    stRecipe.stUCF.iCapSorterTransporterVolumeOfCapsShow.diDefault:=330;
	stRecipe.stUCF.iCapSorterTransporterVolumeOfCapsShow.diMinLimit:=0;
	stRecipe.stUCF.iCapSorterTransporterVolumeOfCapsShow.diMaxLimit:=10000;

    stRecipe.stUCF.iCapSorterWheelWaitingAfterRotationEmptyTableShow.diDefault:=30;
	stRecipe.stUCF.iCapSorterWheelWaitingAfterRotationEmptyTableShow.diMinLimit:=0;
	stRecipe.stUCF.iCapSorterWheelWaitingAfterRotationEmptyTableShow.diMaxLimit:=1000;

    stRecipe.stUCF.iCapSorterWheelWaitingAfterRotationFullTableShow.diDefault:=20;
	stRecipe.stUCF.iCapSorterWheelWaitingAfterRotationFullTableShow.diMinLimit:=0;
	stRecipe.stUCF.iCapSorterWheelWaitingAfterRotationFullTableShow.diMaxLimit:=1000;
	
    stRecipe.stUCF.iCapSorterWheelWaitingAfterRotationHalfFullTableShow.diDefault:=25;
	stRecipe.stUCF.iCapSorterWheelWaitingAfterRotationHalfFullTableShow.diMinLimit:=0;
	stRecipe.stUCF.iCapSorterWheelWaitingAfterRotationHalfFullTableShow.diMaxLimit:=1000;

    stRecipe.stUCF.lrCapSorterBrush1OnWheelPositionHeightSVShow.lrDefault:=20;
	stRecipe.stUCF.lrCapSorterBrush1OnWheelPositionHeightSVShow.lrMinLimit:=0;
	stRecipe.stUCF.lrCapSorterBrush1OnWheelPositionHeightSVShow.lrMaxLimit:=10000;
	
    stRecipe.stUCF.lrCapSorterBrush2OnWheelPositionHeightSVShow.lrDefault:=16;
	stRecipe.stUCF.lrCapSorterBrush2OnWheelPositionHeightSVShow.lrMinLimit:=0;
	stRecipe.stUCF.lrCapSorterBrush2OnWheelPositionHeightSVShow.lrMaxLimit:=10000;

    stRecipe.stUCF.lrCapSorterFeederMover1InputPositionShow.lrDefault:=0;
	stRecipe.stUCF.lrCapSorterFeederMover1InputPositionShow.lrMinLimit:=-10;
	stRecipe.stUCF.lrCapSorterFeederMover1InputPositionShow.lrMaxLimit:=100;
	
	stRecipe.stUCF.lrCapSorterFeederMover1OutputPositionShow.lrDefault:=1147;
	stRecipe.stUCF.lrCapSorterFeederMover1OutputPositionShow.lrMinLimit:=0;
	stRecipe.stUCF.lrCapSorterFeederMover1OutputPositionShow.lrMaxLimit:=1200;
	
    stRecipe.stUCF.lrCapSorterFeederMover2InputPositionShow.lrDefault:=0;
	stRecipe.stUCF.lrCapSorterFeederMover2InputPositionShow.lrMinLimit:=-10;
	stRecipe.stUCF.lrCapSorterFeederMover2InputPositionShow.lrMaxLimit:=100;
	
    stRecipe.stUCF.lrCapSorterFeederMover2OutputPositionShow.lrDefault:=1147;
	stRecipe.stUCF.lrCapSorterFeederMover2OutputPositionShow.lrMinLimit:=0;
    stRecipe.stUCF.lrCapSorterFeederMover2OutputPositionShow.lrMaxLimit:=1200;
	
    stRecipe.stUCF.lrCapSorterFeederMoverAccelerationShow.lrDefault:=60;
	stRecipe.stUCF.lrCapSorterFeederMoverAccelerationShow.lrMinLimit:=0;
	stRecipe.stUCF.lrCapSorterFeederMoverAccelerationShow.lrMaxLimit:=100;
	
    stRecipe.stUCF.lrCapSorterFeederMoverSpeedShow.lrDefault:=50;
	stRecipe.stUCF.lrCapSorterFeederMoverSpeedShow.lrMinLimit:=1;
	stRecipe.stUCF.lrCapSorterFeederMoverSpeedShow.lrMaxLimit:=100;	
	
    stRecipe.stUCF.lrCapSorterFeederSlotDistanceShow.lrDefault:=150;
	stRecipe.stUCF.lrCapSorterFeederSlotDistanceShow.lrMinLimit:=0;
	stRecipe.stUCF.lrCapSorterFeederSlotDistanceShow.lrMaxLimit:=1000;	
	
    stRecipe.stUCF.lrCapSorterIntermediateBrushPositionHeightSVShow.lrDefault:=33;
	stRecipe.stUCF.lrCapSorterIntermediateBrushPositionHeightSVShow.lrMinLimit:=0;
	stRecipe.stUCF.lrCapSorterIntermediateBrushPositionHeightSVShow.lrMaxLimit:=10000;
	
    stRecipe.stUCF.lrCapSorterIntermediateTransporterWheelAngleShow.lrDefault:=3;
	stRecipe.stUCF.lrCapSorterIntermediateTransporterWheelAngleShow.lrMinLimit:=0;
	stRecipe.stUCF.lrCapSorterIntermediateTransporterWheelAngleShow.lrMaxLimit:=360;

    stRecipe.stUCF.lrCapSorterPreScrewerCartesianCatchZPositionShow.lrDefault:=330;
	stRecipe.stUCF.lrCapSorterPreScrewerCartesianCatchZPositionShow.lrMinLimit:=0;
	stRecipe.stUCF.lrCapSorterPreScrewerCartesianCatchZPositionShow.lrMaxLimit:=1000;

    stRecipe.stUCF.lrCapSorterPreScrewerCatcherCatchingPositionShow.lrDefault:=130;
	stRecipe.stUCF.lrCapSorterPreScrewerCatcherCatchingPositionShow.lrMinLimit:=0;
	stRecipe.stUCF.lrCapSorterPreScrewerCatcherCatchingPositionShow.lrMaxLimit:=1000;	
	
    stRecipe.stUCF.lrCapSorterPreScrewerCatcherHightSVShow.lrDefault:=88;
	stRecipe.stUCF.lrCapSorterPreScrewerCatcherHightSVShow.lrMinLimit:=0;
	stRecipe.stUCF.lrCapSorterPreScrewerCatcherHightSVShow.lrMaxLimit:=1000;
	
    stRecipe.stUCF.lrCapSorterPreScrewerCatcherPlacePositionShow.lrDefault:=70;
	stRecipe.stUCF.lrCapSorterPreScrewerCatcherPlacePositionShow.lrMinLimit:=0;
	stRecipe.stUCF.lrCapSorterPreScrewerCatcherPlacePositionShow.lrMaxLimit:=1000;   
	
    stRecipe.stUCF.lrCapSorterPreScrewerCatcherSpeedShow.lrDefault:=20;
	stRecipe.stUCF.lrCapSorterPreScrewerCatcherSpeedShow.lrMinLimit:=1;
	stRecipe.stUCF.lrCapSorterPreScrewerCatcherSpeedShow.lrMaxLimit:=100;  
	
    stRecipe.stUCF.lrCapSorterPreScrewerPickXMover1PositionShow.lrDefault:=188.8;
	stRecipe.stUCF.lrCapSorterPreScrewerPickXMover1PositionShow.lrMinLimit:=0;
	stRecipe.stUCF.lrCapSorterPreScrewerPickXMover1PositionShow.lrMaxLimit:=1000;	
	
    stRecipe.stUCF.lrCapSorterPreScrewerPickXMover2PositionShow.lrDefault:=260;
	stRecipe.stUCF.lrCapSorterPreScrewerPickXMover2PositionShow.lrMinLimit:=0;
	stRecipe.stUCF.lrCapSorterPreScrewerPickXMover2PositionShow.lrMaxLimit:=1000;	
	
    stRecipe.stUCF.lrCapSorterPreScrewerPickZPositionShow.lrDefault:=418;
	stRecipe.stUCF.lrCapSorterPreScrewerPickZPositionShow.lrMinLimit:=0;
	stRecipe.stUCF.lrCapSorterPreScrewerPickZPositionShow.lrMaxLimit:=1000;	
	
	stRecipe.stUCF.lrCapSorterPreScrewerCapCatcherZPositionShow.lrDefault:=450;
	stRecipe.stUCF.lrCapSorterPreScrewerCapCatcherZPositionShow.lrMinLimit:=0;
	stRecipe.stUCF.lrCapSorterPreScrewerCapCatcherZPositionShow.lrMaxLimit:=1000;
	
    stRecipe.stUCF.lrCapSorterPreScrewerPickerSpeedShow.lrDefault:=10;
	stRecipe.stUCF.lrCapSorterPreScrewerPickerSpeedShow.lrMinLimit:=1;
	stRecipe.stUCF.lrCapSorterPreScrewerPickerSpeedShow.lrMaxLimit:=100;	
	
    stRecipe.stUCF.lrCapSorterPreScrewerPlaceXPositionShow.lrDefault:=485.5;
	stRecipe.stUCF.lrCapSorterPreScrewerPlaceXPositionShow.lrMinLimit:=0;
	stRecipe.stUCF.lrCapSorterPreScrewerPlaceXPositionShow.lrMaxLimit:=1000;	
	
    stRecipe.stUCF.lrCapSorterPreScrewerPlaceZPositionShow.lrDefault:=290;
	stRecipe.stUCF.lrCapSorterPreScrewerPlaceZPositionShow.lrMinLimit:=0;
	stRecipe.stUCF.lrCapSorterPreScrewerPlaceZPositionShow.lrMaxLimit:=1000;	
	
    stRecipe.stUCF.lrCapSorterPreScrewerScrewDistanceShow.lrDefault:=360;
	stRecipe.stUCF.lrCapSorterPreScrewerScrewDistanceShow.lrMinLimit:=0;
	stRecipe.stUCF.lrCapSorterPreScrewerScrewDistanceShow.lrMaxLimit:=1400;	
	
    stRecipe.stUCF.lrCapSorterPreScrewerScrewFindingShow.lrDefault:=0;
	stRecipe.stUCF.lrCapSorterPreScrewerScrewFindingShow.lrMinLimit:=0;
	stRecipe.stUCF.lrCapSorterPreScrewerScrewFindingShow.lrMaxLimit:=1000;	
	
    stRecipe.stUCF.lrCapSorterPreScrewerScrewSpeedShow.lrDefault:=50;
	stRecipe.stUCF.lrCapSorterPreScrewerScrewSpeedShow.lrMinLimit:=1;
	stRecipe.stUCF.lrCapSorterPreScrewerScrewSpeedShow.lrMaxLimit:=100;	
	
    stRecipe.stUCF.lrCapSorterPreScrewerScrewerStartZPositionShow.lrDefault:=305;
	stRecipe.stUCF.lrCapSorterPreScrewerScrewerStartZPositionShow.lrMinLimit:=0;
	stRecipe.stUCF.lrCapSorterPreScrewerScrewerStartZPositionShow.lrMaxLimit:=1000;
	
    stRecipe.stUCF.lrCapSorterPreScrewerStrawCatcherZPositionShow.lrDefault:=286;
	stRecipe.stUCF.lrCapSorterPreScrewerStrawCatcherZPositionShow.lrMinLimit:=0;
	stRecipe.stUCF.lrCapSorterPreScrewerStrawCatcherZPositionShow.lrMaxLimit:=1000;
	
    stRecipe.stUCF.lrCapSorterPreScrewerStrawInsertDistance.lrDefault:=50;
	stRecipe.stUCF.lrCapSorterPreScrewerStrawInsertDistance.lrMinLimit:=0;
	stRecipe.stUCF.lrCapSorterPreScrewerStrawInsertDistance.lrMaxLimit:=1000;	
	
    stRecipe.stUCF.lrCapSorterPreScrewerTopZPositionShow.lrDefault:=470;
	stRecipe.stUCF.lrCapSorterPreScrewerTopZPositionShow.lrMinLimit:=0;
	stRecipe.stUCF.lrCapSorterPreScrewerTopZPositionShow.lrMaxLimit:=1000;
	
    stRecipe.stUCF.lrCapSorterRobotPlace1PositionCShow.lrDefault:=0;
	stRecipe.stUCF.lrCapSorterRobotPlace1PositionCShow.lrMinLimit:=-180;
	stRecipe.stUCF.lrCapSorterRobotPlace1PositionCShow.lrMaxLimit:=180;
	
    stRecipe.stUCF.lrCapSorterRobotPlace1PositionXShow.lrDefault:=0;
	stRecipe.stUCF.lrCapSorterRobotPlace1PositionXShow.lrMinLimit:=-100;
	stRecipe.stUCF.lrCapSorterRobotPlace1PositionXShow.lrMaxLimit:=100;
	
    stRecipe.stUCF.lrCapSorterRobotPlace1PositionYShow.lrDefault:=0;
	stRecipe.stUCF.lrCapSorterRobotPlace1PositionYShow.lrMinLimit:=-100;
	stRecipe.stUCF.lrCapSorterRobotPlace1PositionYShow.lrMaxLimit:=100;
	
    stRecipe.stUCF.lrCapSorterRobotPlace1PositionZShow.lrDefault:=20;
	stRecipe.stUCF.lrCapSorterRobotPlace1PositionZShow.lrMinLimit:=-100;
	stRecipe.stUCF.lrCapSorterRobotPlace1PositionZShow.lrMaxLimit:=100;
	
   	stRecipe.stUCF.lrCapSorterWheelMoveAngleEmptyTableShow.lrDefault:=16;
	stRecipe.stUCF.lrCapSorterWheelMoveAngleEmptyTableShow.lrMinLimit:=0;
	stRecipe.stUCF.lrCapSorterWheelMoveAngleEmptyTableShow.lrMaxLimit:=360;
	
    stRecipe.stUCF.lrCapSorterWheelMoveAngleFullyTableShow.lrDefault:=1;
	stRecipe.stUCF.lrCapSorterWheelMoveAngleFullyTableShow.lrMinLimit:=0;
	stRecipe.stUCF.lrCapSorterWheelMoveAngleFullyTableShow.lrMaxLimit:=360;
	
    stRecipe.stUCF.lrCapSorterWheelMoveAngleHalfFullyTableShow.lrDefault:=6;
	stRecipe.stUCF.lrCapSorterWheelMoveAngleHalfFullyTableShow.lrMinLimit:=0;
	stRecipe.stUCF.lrCapSorterWheelMoveAngleHalfFullyTableShow.lrMaxLimit:=360;
	
    stRecipe.stUCF.udiCapSorterIntermediateTransporterTimeProductOnSensorShow.udiDefault:=800;
	stRecipe.stUCF.udiCapSorterIntermediateTransporterTimeProductOnSensorShow.udiMinLimit:=0;
	stRecipe.stUCF.udiCapSorterIntermediateTransporterTimeProductOnSensorShow.udiMaxLimit:=10000;
	
    stRecipe.stUCF.udiCapSorterTransporterTimeProductOnSensorBeforeBrushShow.udiDefault:=110;
	stRecipe.stUCF.udiCapSorterTransporterTimeProductOnSensorBeforeBrushShow.udiMinLimit:=0;
	stRecipe.stUCF.udiCapSorterTransporterTimeProductOnSensorBeforeBrushShow.udiMaxLimit:=10000;
	
    stRecipe.stUCF.uiCapSorterIndexShow.udiDefault:=8;
	stRecipe.stUCF.uiCapSorterIndexShow.udiMinLimit:=1;
	stRecipe.stUCF.uiCapSorterIndexShow.udiMaxLimit:=100000;
	
	stRecipe.stUCF.lrCapSorterWheelMoveDecelerationEmptyTableShow.lrDefault:=4000;//nie używane
	
	stRecipe.stUCF.lrCapSorterWheelMoveDecelerationFullTableShow.lrDefault:=4000;//nie używane
	
	stRecipe.stUCF.lrCapSorterWheelMoveDecelerationHalfFullTableShow.lrDefault:=4000;//nie używane
	
	stRecipe.stUCF.lrCapSorterWheelMoveSpeedEmptyTableShow.lrDefault:=300;//nie używane
	
	stRecipe.stUCF.lrCapSorterWheelMoveSpeedFullTableShow.lrDefault:=300;//nie używane
	
	stRecipe.stUCF.lrCapSorterWheelMoveSpeedHalfFullTableShow.lrDefault:=300;//nie używane
	
	stRecipe.stUCF.lrCapSorterWheelJerkAngleEmptyTableShow.lrDefault:=10000;//nie używane
	
	stRecipe.stUCF.lrCapSorterWheelJerkAngleFullTableShow.lrDefault:=14000;//nie używane
	
	stRecipe.stUCF.lrCapSorterWheelJerkAngleHalfFullTableShow.lrDefault:=14000;//nie używane
	
	stRecipe.stUCF.lrCapSorterWheelMoveAccelerationEmptyTableShow.lrDefault:=4000;//nie używane
	
	stRecipe.stUCF.lrCapSorterWheelMoveAccelerationFullTableShow.lrDefault:=4000;//nie używane
	
	stRecipe.stUCF.lrCapSorterWheelMoveAccelerationHalfFullTableShow.lrDefault:=4000;//nie używane
	
    stRecipe.stUCF.lrCapSorterPreScrewerScrewJerkShow.lrDefault:=350000;//nie używane
	
	stRecipe.stUCF.lrCapSorterPreScrewerScrewAccelerationShow.lrDefault:=30000;//nie używane
	
	stRecipe.stUCF.lrCapSorterPreScrewerPickerAccelerationShow.lrDefault:=30000;//nie używane
	
	stRecipe.stUCF.lrCapSorterPreScrewerPickerJerkShow.lrDefault:=100000;//nie używane	
	
	stRecipe.stUCF.lrCapSorterPreScrewerGripperOpenPositionShow.lrDefault:=275;//nie używane
	
	stRecipe.stUCF.lrCapSorterPreScrewerCatcherReleseShow.lrDefault:=240;//nie używane
	
	stRecipe.stUCF.lrCapSorterPreScrewerCatcherJerkShow.lrDefault:=100000;//nie używane
	
	stRecipe.stUCF.lrCapSorterPreScrewerCatchAngleOpenSV.lrDefault:=180;//nie używane w ekranie receptur
	
	stRecipe.stUCF.lrCapSorterPreScrewerCatcherAccelerationShow.lrDefault:=40000;// nie używane
	
	stRecipe.stUCF.lrCapSorterPreScrewerBendingDistanceShow.lrDefault:=10;//nie używane
	
	stRecipe.stUCF.lrCapSorterPreScrewerBottleCatch1CloseValueShow.lrDefault:=20600;//nie używane
	
	stRecipe.stUCF.lrCapSorterPreScrewerBottleCatch1OpenValueShow.lrDefault:=43110;//nie używane
	
	stRecipe.stUCF.lrCapSorterPreScrewerBottleCatch2CloseValueShow.lrDefault:=23300;//nie używane
	
	stRecipe.stUCF.lrCapSorterPreScrewerBottleCatch2OpenValueShow.lrDefault:=45548;//nie używane
	
	stRecipe.stUCF.lrCapSorterPreScrewerBottleCatch3CloseValueShow.lrDefault:=21200;//nie uzywane
	
	stRecipe.stUCF.lrCapSorterPreScrewerBottleCatch3OpenValueShow.lrDefault:=44110;//nie używane
	
	stRecipe.stUCF.lrCapSorterPreScrewerBottleCatch4CloseValueShow.lrDefault:=19500;//nie używane
	
	stRecipe.stUCF.lrCapSorterPreScrewerBottleCatch4OpenValueShow.lrDefault:=42487;//nie używane
	
	stRecipe.stUCF.lrCapSorterFeederMoveJerkShow.lrDefault:=370000;//nie używane
	
	stRecipe.stUCF.iCapSorterRobotGripperWatchdogShow.diDefault:=10;//nie używane
	
	stRecipe.stUCF.iCapSorterRobotNumberToolShow.diDefault:=0;//nie używane
	
	stRecipe.stUCF.iCapSorterRobotParalaxCorrectionShow.diDefault:=0;//nie używane
	
	stRecipe.stUCF.iCapSorterIntermediateTransporterManualSpeedShow.diDefault:=30;//nie używane
	
	stRecipe.stUCF.iCapSorterIntermediateBrushManualSpeedShow.diDefault:=30;//nie używane
	
	stRecipe.stUCF.iCapSorterBrush2OnWheelManualSpeedShow.diDefault:=20;//nie używane
	
	stRecipe.stUCF.iCapSorterBrush1OnWheelManualSpeedShow.diDefault:=30;//nie używane
	
	stRecipe.stUCF.lrCapSorterPreScrewerWaitInPlaceTimeShow.lrDefault:=50;//nie używane
	
	stRecipe.stUBF.lrBottleSorterZPickAboveTheBottleSVShow.lrDefault:=0;// nie używane

	stRecipe.stUBF.lrBottleSorterZPickMoveSVShow.lrDefault:=0;// nie używane

	stRecipe.stUBF.uiBottleSorterIndexShow.diDefault:=0;// nie używane
	
	stRecipe.stUBF.lrBottleSorterRemainingTimeToRejectShow.lrDefault:=0;//nie używane
	
	stRecipe.stUBF.lrBottleSorterRemainingTimeToSuctionShow.lrDefault:=0;// nie używane
	
	stRecipe.stUBF.lrBottleSorterSafetyHeightSVShow.lrDefault:=0;// nie używane
	
	stRecipe.stUBF.lrBottleSorterSuckerSuctionTimeShow.lrDefault:=0;// nie używane
	
	stRecipe.stUBF.lrBottleSorterEjectorPulseShow.lrDefault:=0;//nie używane
	
	stRecipe.stUBF.iBottleSorterSupplyTimeThirdConditionSVShow.diDefault:=0;//nie używane
	
	stRecipe.stUBF.iBottleSorterSensorsCountSecondConditionMinSVShow.diDefault:=0;//nie używane
	
	stRecipe.stUBF.iBottleSorterSensorsCountThirdConditionSVShow.diDefault:=0;//nie używane
	
	stRecipe.stUBF.iBottleSorterProductTypeShow.diDefault:=0; //nie używane
	
	stRecipe.stUBL.iLidPuttedCheckProgramShow.diDefault:=0;// nie używane
	
	stRecipe.stUBL.iCapFeederGateBlockingTimeShow.diDefault:=100;// nie używane	
	
    stRecipe.stUBL.iWeight1ActuatorUpDelayShow.diDefault:=0;//nie używane
	
    stRecipe.stUBL.iWeight2ActuatorUpDelayShow.diDefault:=0;//nie używane
	
    stRecipe.stUBL.iWeight3ActuatorUpDelayShow.diDefault:=0;//nie używane
	
    stRecipe.stUBL.iWeight4ActuatorUpDelayShow.diDefault:=0;//nie używane	
	
    stRecipe.stUBL.iWeight5ActuatorUpDelayShow.diDefault:=0;//nie używane	
	
    stRecipe.stUBL.iWeight6ActuatorUpDelayShow.diDefault:=0;//nie używane
	
	stRecipe.stUBL.lrDispencer1SuckValveCloseVolumeShow.lrDefault:=0;//nie używane
	
	stRecipe.stUBL.lrDispencer1DoseValveOpenVolumeShow.lrDefault:=0;//nie używane
	
    stRecipe.stUBL.lrDispencer1LifterAccelerationShow.lrDefault:=15000;//nie używane
	
    stRecipe.stUBL.lrDispencer1LifterDecelerationShow.lrDefault:=15000;//nie używane
	
	stRecipe.stUBL.lrDispencer1LifterVelocityShow.lrDefault:=1050;//nie używane
	
	stRecipe.stUBL.lrDispencer2DoseValveOpenVolumeShow.lrDefault:=0;// nie używane
	
	stRecipe.stUBL.lrDispencer2LifterAccelerationShow.lrDefault:=15000;//nie używane

	stRecipe.stUBL.lrDispencer2LifterDecelerationShow.lrDefault:=15000;//nie używane
		
    stRecipe.stUBL.lrDispencer2LifterVelocityShow.lrDefault:=1050;// nie używane
	
	stRecipe.stUBL.lrDispencer2SuckValveCloseVolumeShow.lrDefault:=0;// nie używane	
	
    stRecipe.stUBL.lrFormWeightShow.lrDefault:=0;//nie używane
	
    stRecipe.stUBL.lrGripperScrewerPressureExhaustLevelShow.lrDefault:=100;//nie używane
		
    stRecipe.stUBL.lrGripperScrewerCatchPressureExhaustLevelShow.lrDefault:=100;//nie używane
	
    stRecipe.stUBL.lrLidPuttedCheckAreaShow.lrDefault:=200;//nie używane
	
    stRecipe.stUBL.lrLidPuttedCheckHeightSVShow.lrDefault:=200;//nie używane
	
    stRecipe.stUBL.lrLidPuttedCheckPositionShow.lrDefault:=200;//nie używane
	
    stRecipe.stUBL.lrMass1DensityShow.lrDefault:=1;//nie używane
	
    stRecipe.stUBL.lrMass2DensityShow.lrDefault:=1;//nie używane
	
    stRecipe.stUBL.lrWeight1MeasurmentCorrectionShow.lrDefault:=0;//nie używane
		
    stRecipe.stUBL.lrWholePackageWeightShow.lrDefault:=0;//nie używane
	
    stRecipe.stUBL.nBottleTransferProgramShow.udiDefault:=0;//nie używane
		
    stRecipe.stUBL.nFormTransportersSlowerVelocitySVShow.udiDefault:=1800;//nie używane
	
    stRecipe.stUBL.nGateAfterWeightTimeFormInsertingShow.lrDefault:=250;//nie używane
	
    stRecipe.stUBL.nGateBeforeDispencersTimeFormInsertingShow.lrDefault:=300;//nie używane
	
    stRecipe.stUBL.nGateRobotTimeFormInsertingShow.lrDefault:=250;//nie używane
END_IF
METH_SortRecipesTable(0);
		udiCurrentIndex																		:=	0;
		wsCurrentCaption1																	:=	"Factory defaults";
		wsCurrentCaption2																	:=	"-";
		METH_SetFactoryDefaults(stPrcRecipe:=stActRecipe);
		udiInitCase										:=	1000;

	1000:
		;

END_CASE
END_ACTION

ACTION ACT_LoadRecipe:
CASE iLoadRecipeCase OF
	0:
				bRecipeLoaded						:=FALSE;
	10:
		IF (iSelectedArrayIndex >=0) THEN 
			IF (aRecipeList[iSelectedArrayIndex].wsRecipeCaption <>"") THEN
				diFileLoadIndex						:=	aRecipeList[iSelectedArrayIndex].udiIndex;
				fbRecipeLoad.sFilePath				:=	CONCAT(CONCAT('C:\Recipes\',DINT_TO_STRING(diFileLoadIndex)),'.CSV');
				fbRecipeLoad.database				:= 	ADR(aRecipeParamsValues);
				fbRecipeLoad.nRows					:= 	udiMaxParamsVariablesCount;
				fbRecipeLoad.nCols					:= 	0;	
				fbRecipeLoad.bExecute				:=	TRUE;
				iLoadRecipeCase						:=	20;
			ELSE
				iLoadRecipeCase				:=	0;
			END_IF
		ELSE
			iLoadRecipeCase					:=	0;
		END_IF
		
	20:
		IF (fbRecipeLoad.bError) THEN
			fbRecipeLoad.bExecute			:=	FALSE;
			iLoadRecipeCase					:=	0;
		END_IF
		IF (fbRecipeLoad.bDone) THEN
			METH_FileStructToRecipeStuct();
			
			wsCurrentCaption1				:=	aRecipeList[diSelectedRecipeFileArrayIndex].wsRecipeCaption;
			wsCurrentCaption2				:=	aRecipeList[diSelectedRecipeFileArrayIndex].wsRecipeDescription;
			udiCurrentIndex					:=	aRecipeList[diSelectedRecipeFileArrayIndex].udiIndex;
			
			fbRecipeLoad.bExecute			:=	FALSE;
			iLoadRecipeCase					:=	0;
			
			bRecipeLoaded					:=	TRUE;
			
			P030_Recipes.bShowRecipeHomingWarning	:=TRUE;
		END_IF
END_CASE
END_ACTION

ACTION ACT_RenameRecipe:
CASE iRenameRecipeCase OF
	0:
		;
	10:
		
		fbRecipeRename.sNetId				:=	'';
		fbRecipeRename.sOldName				:=	CONCAT(CONCAT('C:\Recipes\',UDINT_TO_STRING(udiEditOldIndex)),'.CSV');
		fbRecipeRename.sNewName				:=	CONCAT(CONCAT('C:\Recipes\',UDINT_TO_STRING(udiEditNewIndex)),'.CSV');
		fbRecipeRename.ePath				:= 	PATH_GENERIC;
		fbRecipeRename.tTimeout				:= 	T#3S;
		fbRecipeRename.bExecute				:=	TRUE;
		iRenameRecipeCase					:=	20;
	20:
		IF (fbRecipeRename.bError) THEN
			fbRecipeRename.bExecute			:=	FALSE;
			bEditFail						:=	TRUE;
			wsEditErrorMessage				:=	"Nie udało się zapisać pliku";			
			iRenameRecipeCase				:=	0;
		ELSIF NOT fbRecipeRename.bBusy THEN
			bEditOk							:=	TRUE;
			fbRecipeRename.bExecute			:=	FALSE;
			iRenameRecipeCase				:=	0;			
		END_IF
		
END_CASE
END_ACTION

ACTION ACT_SaveRecipe:
CASE iSaveRecipeCase OF
	0:
		;
	10:
		fbRecipeSave.sFilePath				:=	CONCAT(CONCAT('C:\Recipes\',DINT_TO_STRING(diFileSaveIndex)),'.CSV');
//		fbRecipeSave.database				:= 	ADR(aRecipeParamsValues);
		fbRecipeSave.nRows					:= 	udiMaxParamsVariablesCount;
		fbRecipeSave.nCols					:= 	0;
		fbRecipeSave.bExecute				:=	TRUE;
		iSaveRecipeCase						:=	20;
	20:
		IF (fbRecipeSave.bError OR fbRecipeSave.bDone) THEN
			fbRecipeSave.bExecute			:=	FALSE;
			iSaveRecipeCase					:=	0;
		END_IF
END_CASE
END_ACTION

ACTION ACT_UpdateList:
CASE udiUpdateCase OF
	0:
		;
	10: 
		diRecipeCaptionMaxIndex									:=	-1;
		FOR i:=0 TO udiMaxRecipeCount DO
			IF (aRecipeList[i].bUsed) THEN
				diRecipeCaptionMaxIndex							:=	diRecipeCaptionMaxIndex +1;
//				aRecipeIndexArray[diRecipeCaptionMaxIndex]		:=	UDINT_TO_DINT(i);
				aRecipeCaptionArray[0,diRecipeCaptionMaxIndex]	:=	UDINT_TO_WSTRING(aRecipeList[i].udiIndex);
				aRecipeCaptionArray[1,diRecipeCaptionMaxIndex]	:=	aRecipeList[i].wsRecipeCaption;
				aRecipeCaptionArray[2,diRecipeCaptionMaxIndex]	:=	aRecipeList[i].wsCreateDate;		
			END_IF
		END_FOR
		
		FOR i := DINT_TO_UDINT(diRecipeCaptionMaxIndex +1) TO udiMaxRecipeCount DO
				aRecipeCaptionArray[0,i]						:=	"";
				aRecipeCaptionArray[1,i]						:=	"";
				aRecipeCaptionArray[2,i]						:=	"";	
		END_FOR
		METH_CreateRecipesListStringArray();
		METH_SortRecipesTable(0);
		udiUpdateCase									:=	20;	
	20:
		fbListSave.bExecute								:=	TRUE;
		udiUpdateCase									:=	30;
	30:
		IF (fbListSave.bDone) THEN
			fbListSave.bExecute							:=	FALSE;
			udiUpdateCase								:=	0;
		END_IF
		IF (fbListSave.bError) THEN
			fbListSave.bExecute							:=	FALSE;
			udiUpdateCase								:=	0;
		END_IF

END_CASE

IF bLineSelect THEN
	diSelectedRecipeFileArrayIndex						:= 	METH_FindRecipeArrayIndex(iSelectedArrayIndex);
	wsSelectedCaption									:= 	aRecipeList[diSelectedRecipeFileArrayIndex].wsRecipeCaption;
	udiSelectedRecipeIndex								:=	aRecipeList[diSelectedRecipeFileArrayIndex].udiIndex;	
	bLineSelect											:= 	FALSE;
	
	sProductBitmapId									:= CONCAT('C:\Recipe_photos\RecipeImages.',UDINT_TO_STRING(udiSelectedRecipeIndex));
	sProductBitmapId									:=Concat(sProductBitmapId,'.jpg');
	
END_IF
END_ACTION

METHOD METH_CreateOrClone : BOOL
VAR_INPUT
	bSetDefault				:	BOOL;	
END_VAR
VAR 
	aiCreateDate										:	ARRAY[0..5] OF UINT;
END_VAR

	bAlreadyExist										:=	FALSE;
	bNewRecipeError										:=	FALSE;
	
	IF (wsNewRecipeCaption = "") THEN
		bNewRecipeError									:=	TRUE;
		wsNewRecipeError								:=	"Nazwa nie może być pusta";
	ELSE
		FOR i:= 0 TO udiMaxRecipeCount DO
			IF (aRecipeList[i].bUsed AND (aRecipeList[i].wsRecipeCaption = wsNewRecipeCaption OR aRecipeList[i].udiIndex = udiNewRecipeIndex)) THEN 
				bAlreadyExist							:=	TRUE;
				EXIT;
			END_IF
		END_FOR
		IF (bAlreadyExist) THEN
			bNewRecipeError								:=	TRUE;
			wsNewRecipeError							:=	"Receptura z taką nazwą lub indeksem była dodana wcześnej";
		ELSIF (iSaveRecipeCase >0 OR udiUpdateCase > 0) THEN
			bNewRecipeError								:=	TRUE;
			wsNewRecipeError							:=	"Błąd tworzenia pliku";
		ELSE
			FOR i:= 0 TO udiMaxRecipeCount DO
				IF (NOT aRecipeList[i].bUsed) THEN
					aRecipeList[i].bUsed				:=	TRUE;
					aRecipeList[i].wsRecipeCaption		:=	wsNewRecipeCaption;
					aRecipeList[i].wsRecipeDescription	:=	wsNewRecipeDescription;
					aRecipeList[i].udiIndex				:=	udiNewRecipeIndex;
					
					aiCreateDate[0]		:=	P020_RtcEffectivityOEE.stActualTime.wYear;
					aiCreateDate[1]		:=	P020_RtcEffectivityOEE.stActualTime.wMonth;
					aiCreateDate[2]		:=	P020_RtcEffectivityOEE.stActualTime.wDay;
					aiCreateDate[3]		:=	P020_RtcEffectivityOEE.stActualTime.wHour;
					aiCreateDate[4]		:=	P020_RtcEffectivityOEE.stActualTime.wMinute;
					aiCreateDate[5]		:=	P020_RtcEffectivityOEE.stActualTime.wSecond;
					
					aRecipeList[i].wsCreateDate 		:= METH_DateTimeArray_To_Wstring(aiCreateDate);
					
					IF (bSetDefault) THEN
						METH_SetFactoryDefaults(stPrcRecipe:=stActRecipe);
					END_IF
					METH_RecipeStuctToFileStruct();
					METH_SortRecipesTable(0);				
					diFileSaveIndex						:=	UDINT_TO_INT(udiNewRecipeIndex);
					iSaveRecipeCase						:=	10;
					udiUpdateCase						:=	10;
	
					bNewRecipeOk						:=	TRUE;
					wsNewRecipeError					:=	"";
					EXIT;
				END_IF
			END_FOR
			IF (NOT bNewRecipeOk) THEN
				bNewRecipeError							:=	TRUE;
				wsNewRecipeError						:=	"Nie ma wolnego miejsca w tabeli receptur";
			END_IF
		END_IF
	END_IF
END_METHOD

METHOD METH_CreateRecipesListStringArray : BOOL
VAR

END_VAR

FOR i := 0 TO udiMaxRecipeCount DO
	aRecipeListString[i] := BOOL_TO_STRING(aRecipeList[i].bUsed);
	aRecipeListString[i] := CONCAT(aRecipeListString[i],'|');	
	aRecipeListString[i] := CONCAT(aRecipeListString[i],UDINT_TO_STRING(aRecipeList[i].udiIndex));
	aRecipeListString[i] := CONCAT(aRecipeListString[i],'|');
	aRecipeListString[i] := CONCAT(aRecipeListString[i],WSTRING_TO_STRING(aRecipeList[i].wsRecipeCaption));
	aRecipeListString[i] := CONCAT(aRecipeListString[i],'|');
	aRecipeListString[i] := CONCAT(aRecipeListString[i],WSTRING_TO_STRING(aRecipeList[i].wsRecipeDescription));
	aRecipeListString[i] := CONCAT(aRecipeListString[i],'|');
	aRecipeListString[i] := CONCAT(aRecipeListString[i],WSTRING_TO_STRING(aRecipeList[i].wsCreateDate));
END_FOR
END_METHOD

METHOD METH_DateTimeArray_To_Wstring : WSTRING
VAR_INPUT
	aDate	:	ARRAY[0..5] OF UINT;
END_VAR
VAR 
	wsTmp												:	WSTRING;
END_VAR
IF (aDate[2]<10) THEN
	wsTmp:="0";
END_IF
wsTmp:=WCONCAT(wsTmp,WCONCAT(UINT_TO_WSTRING(aDate[2]),"."));
IF (aDate[1]<10) THEN
	wsTmp:=WCONCAT(wsTmp,"0");
END_IF
wsTmp:=WCONCAT(wsTmp,WCONCAT(UINT_TO_WSTRING(aDate[1]),"."));

IF (aDate[0]<1000) THEN
	wsTmp:=WCONCAT(wsTmp,"0");
ELSIF (aDate[0]<100) THEN
	wsTmp:=WCONCAT(wsTmp,"00");
ELSIF (aDate[0]<10) THEN
	wsTmp:=WCONCAT(wsTmp,"000");
END_IF
wsTmp:=WCONCAT(wsTmp,WCONCAT(UINT_TO_WSTRING(aDate[0])," "));

IF (aDate[3]<10) THEN
	wsTmp:=WCONCAT(wsTmp,"0");
END_IF
wsTmp:=WCONCAT(wsTmp,WCONCAT(UINT_TO_WSTRING(aDate[3]),":"));
IF (aDate[4]<10) THEN
	wsTmp:=WCONCAT(wsTmp,"0");
END_IF
wsTmp:=WCONCAT(wsTmp,WCONCAT(UINT_TO_WSTRING(aDate[4]),"."));
IF (aDate[5]<10) THEN
	wsTmp:=WCONCAT(wsTmp,"0");
END_IF
wsTmp:=WCONCAT(wsTmp,UINT_TO_WSTRING(aDate[5]));
METH_DateTimeArray_To_Wstring:=wsTmp;
END_METHOD

METHOD METH_Edit : BOOL
VAR_INPUT
END_VAR
bEditFail											:=	FALSE;
bEditOk												:=	FALSE;

IF (wsEditNewCaption1 = "") THEN
	bEditFail										:=	TRUE;
	wsEditErrorMessage								:=	"Nazwa nie może być pustą";
ELSE
	FOR i:= 0 TO udiMaxRecipeCount DO
		IF (
			aRecipeList[i].bUsed AND 
			(aRecipeList[i].wsRecipeCaption = wsEditNewCaption1 OR aRecipeList[i].udiIndex =udiEditNewIndex) (*udiEditNewIndex)*) AND
			diSelectedRecipeFileArrayIndex <> UDINT_TO_DINT(i)
			) THEN 
			bEditFail								:=	TRUE;
			wsEditErrorMessage						:=	"Receptura z taką nazwą lub indeksem była dodana wcześniej";	
			RETURN;
		END_IF
	END_FOR
	
	IF (iSelectedArrayIndex >=0) THEN
		IF (diSelectedRecipeFileArrayIndex>=0) THEN
			udiEditOldIndex 													:= 	aRecipeList[diSelectedRecipeFileArrayIndex].udiIndex;
			aRecipeList[diSelectedRecipeFileArrayIndex].udiIndex				:=	udiEditNewIndex;
			aRecipeList[diSelectedRecipeFileArrayIndex].wsRecipeCaption			:=	wsEditNewCaption1;
			aRecipeList[diSelectedRecipeFileArrayIndex].wsRecipeDescription		:=	wsEditNewCaption2;
			IF (udiUpdateCase = 0) THEN
				udiUpdateCase						:=	10;
			END_IF
			IF udiEditOldIndex <> udiEditNewIndex AND iRenameRecipeCase = 0 THEN
				iRenameRecipeCase 					:= 	10;
			END_IF
		END_IF
	END_IF
	IF NOT bEditFail AND iRenameRecipeCase = 0 THEN
		bEditOk											:=	TRUE;		
	END_IF

END_IF
END_METHOD

METHOD METH_FileStructToRecipeStuct : BOOL
VAR_INPUT
END_VAR

VAR
END_VAR
stActRecipe.stUBL.nRecipeIndexShow.diValue															:=						STRING_TO_DINT	(aRecipeParamsValues[0  ]);
stActRecipe.stUBL.iPackageCapTypeShow.diValue														:=						STRING_TO_DINT	(aRecipeParamsValues[1  ]);		
stActRecipe.stUBL.iPackageCapDiameterShow.diValue 													:=						STRING_TO_DINT	(aRecipeParamsValues[2  ]);       
stActRecipe.stUBL.bExEnableShow.bValue 																:=						STRING_TO_BOOL	(aRecipeParamsValues[3  ]);
stActRecipe.stUBL.bBottleFeederEnableShow.bValue													:=						STRING_TO_BOOL	(aRecipeParamsValues[4  ]);
stActRecipe.stUBL.iBottleFeederTurntableVelocitySVShow.udiValue										:=						STRING_TO_UDINT (aRecipeParamsValues[5  ]);
stActRecipe.stUBL.iBottleFeederBottleSensorDelayShow.diValue										:=						STRING_TO_DINT	(aRecipeParamsValues[6  ]);
stActRecipe.stUBL.iBottleFeederFormGateDelayShow.diValue											:=						STRING_TO_DINT	(aRecipeParamsValues[7  ]);
stActRecipe.stUBL.iBottleFeederAllowFormDelayShow.diValue											:=						STRING_TO_DINT	(aRecipeParamsValues[8  ]);
stActRecipe.stUBL.bPucksInserterEnableShow.bValue													:=						STRING_TO_BOOL	(aRecipeParamsValues[9  ]); 
stActRecipe.stUBL.iPucksInserterTurntableVelocitySVShow.udiValue 									:=						STRING_TO_UDINT (aRecipeParamsValues[10 ]);  
stActRecipe.stUBL.iPucksInserterConveyorVelocitySVShow.udiValue										:=						STRING_TO_UDINT (aRecipeParamsValues[11 ]); 
stActRecipe.stUBL.iPucksInserterBottleSensorDelayShow.diValue										:=						STRING_TO_DINT	(aRecipeParamsValues[12 ]);
stActRecipe.stUBL.iPucksInserterFormGateDelayShow.diValue 											:=						STRING_TO_DINT	(aRecipeParamsValues[13 ]);
stActRecipe.stUBL.iPucksInserterAllowFormDelayShow.diValue 											:=						STRING_TO_DINT	(aRecipeParamsValues[14 ]);
stActRecipe.stUBL.lrPucksInserterWheelOffsetShow.lrValue 											:=						STRING_TO_LREAL (aRecipeParamsValues[15 ]);
stActRecipe.stUBL.lrPucksInserterWheelAccelerationShow.lrValue 										:=						STRING_TO_LREAL (aRecipeParamsValues[16 ]);
stActRecipe.stUBL.lrPucksInserterWheelVelocityShow.lrValue 											:=						STRING_TO_LREAL (aRecipeParamsValues[17 ]);
stActRecipe.stUBL.lrPucksInserterHammerHeightSVShow.lrValue 										:=						STRING_TO_LREAL (aRecipeParamsValues[18 ]);
stActRecipe.stUBL.bGateBeforeDispencersEnableShow.bValue											:=						STRING_TO_BOOL	(aRecipeParamsValues[19 ]);
stActRecipe.stUBL.nGateBeforeDispencersTimeFormInsertingShow.lrValue 								:=						STRING_TO_LREAL (aRecipeParamsValues[20 ]);
stActRecipe.stUBL.bGateAfterWeightEnableShow.bValue 												:=						STRING_TO_BOOL	(aRecipeParamsValues[21 ]);
stActRecipe.stUBL.nGateAfterWeightTimeFormInsertingShow.lrValue 									:=						STRING_TO_LREAL (aRecipeParamsValues[22 ]);
stActRecipe.stUBL.bGateRobotEnableShow.bValue       												:=						STRING_TO_BOOL	(aRecipeParamsValues[25 ]);
stActRecipe.stUBL.nGateRobotTimeFormInsertingShow.lrValue											:=						STRING_TO_LREAL (aRecipeParamsValues[26 ]);
stActRecipe.stUBL.bFormsDragingLeftEnableShow.bValue         										:=						STRING_TO_BOOL	(aRecipeParamsValues[27 ]);
stActRecipe.stUBL.lrFormsDragingLeftVelocityShow.lrValue         									:=						STRING_TO_LREAL (aRecipeParamsValues[28 ]);
stActRecipe.stUBL.lrFormsDragingLeftAccelerationShow.lrValue 										:=						STRING_TO_LREAL (aRecipeParamsValues[29 ]);
stActRecipe.stUBL.lrFormsDragingLeftDecelerationShow.lrValue   										:=						STRING_TO_LREAL (aRecipeParamsValues[30 ]);
stActRecipe.stUBL.bFormsDragingRightEnableShow.bValue 												:=						STRING_TO_BOOL	(aRecipeParamsValues[31 ]);
stActRecipe.stUBL.lrFormsDragingRightVelocityShow.lrValue 											:=						STRING_TO_LREAL (aRecipeParamsValues[32 ]);
stActRecipe.stUBL.lrFormsDragingRightAccelerationShow.lrValue 										:=						STRING_TO_LREAL (aRecipeParamsValues[33 ]);
stActRecipe.stUBL.lrFormsDragingRightDecelerationShow.lrValue 										:=						STRING_TO_LREAL (aRecipeParamsValues[34 ]);
stActRecipe.stUBL.bDosingTwoPhasesShow.bValue 	        											:=						STRING_TO_BOOL	(aRecipeParamsValues[35 ]);
stActRecipe.stUBL.lrDispencersLifterReadyPositionShow.lrValue 										:=						STRING_TO_LREAL (aRecipeParamsValues[36 ]);
stActRecipe.stUBL.uiDispencerStartDosingDelayShow.udiValue 											:=						STRING_TO_UDINT (aRecipeParamsValues[37 ]);
stActRecipe.stUBL.bDispencer1EnableShow.bValue 	          											:=						STRING_TO_BOOL	(aRecipeParamsValues[38 ]);
stActRecipe.stUBL.bDispencer2EnableShow.bValue 		  												:=						STRING_TO_BOOL	(aRecipeParamsValues[39 ]);
stActRecipe.stUBL.bDispencer3EnableShow.bValue           											:=						STRING_TO_BOOL	(aRecipeParamsValues[40 ]);
stActRecipe.stUBL.bDispencer4EnableShow.bValue 			       										:=						STRING_TO_BOOL	(aRecipeParamsValues[41 ]);
stActRecipe.stUBL.lrDispencer1DoseVolumeShow.lrValue 				   								:=						STRING_TO_LREAL (aRecipeParamsValues[42 ]);
stActRecipe.stUBL.lrDispencer1Phase1VolumeShow.lrValue	           									:=						STRING_TO_LREAL (aRecipeParamsValues[43 ]);
stActRecipe.stUBL.lrDispencer1Phase2VolumeShow.lrValue 	       										:=						STRING_TO_LREAL (aRecipeParamsValues[44 ]);
stActRecipe.stUBL.lrDispencer1Phase1VelocityShow.lrValue 	       									:=						STRING_TO_LREAL (aRecipeParamsValues[45 ]);
stActRecipe.stUBL.lrDispencer1Phase2VelocityShow.lrValue 											:=						STRING_TO_LREAL (aRecipeParamsValues[46 ]);
stActRecipe.stUBL.lrDispencer1Phase3VelocityShow.lrValue 		   									:=						STRING_TO_LREAL (aRecipeParamsValues[47 ]);
stActRecipe.stUBL.lrDispencer1SuckVelocityShow.lrValue   											:=						STRING_TO_LREAL (aRecipeParamsValues[48 ]);
stActRecipe.stUBL.lrDispencer1Phase1AccelerationShow.lrValue 										:=						STRING_TO_LREAL (aRecipeParamsValues[49 ]);
stActRecipe.stUBL.lrDispencer1Phase2AccelerationShow.lrValue 	  									:=						STRING_TO_LREAL (aRecipeParamsValues[50 ]);
stActRecipe.stUBL.lrDispencer1Phase3AccelerationShow.lrValue 	   									:=						STRING_TO_LREAL (aRecipeParamsValues[51 ]);
stActRecipe.stUBL.lrDispencer1SuckAccelerationShow.lrValue  										:=						STRING_TO_LREAL (aRecipeParamsValues[52 ]);
stActRecipe.stUBL.lrDispencer1Phase1DecelerationShow.lrValue        								:=						STRING_TO_LREAL (aRecipeParamsValues[53 ]);
stActRecipe.stUBL.lrDispencer1Phase2DecelerationShow.lrValue 										:=						STRING_TO_LREAL (aRecipeParamsValues[54 ]);
stActRecipe.stUBL.lrDispencer1Phase3DecelerationShow.lrValue 	   									:=						STRING_TO_LREAL (aRecipeParamsValues[55 ]);
stActRecipe.stUBL.udiDispencer1DosingDoneDelayTimeShow.udiValue 									:=						STRING_TO_UDINT (aRecipeParamsValues[56 ]);
stActRecipe.stUBL.lrDispencer1SuckValveOpenVolumeShow.lrValue 										:=						STRING_TO_LREAL (aRecipeParamsValues[57 ]);
stActRecipe.stUBL.lrDispencer1SuckValveOpenTimeDelayShow.lrValue 									:=						STRING_TO_LREAL (aRecipeParamsValues[58 ]);
stActRecipe.stUBL.lrDispencer1SuckValveCloseVolumeShow.lrValue 										:=						STRING_TO_LREAL (aRecipeParamsValues[59 ]);
stActRecipe.stUBL.lrDispencer1SuckValveCloseTimeDelayShow.lrValue 									:=						STRING_TO_LREAL (aRecipeParamsValues[60 ]);
stActRecipe.stUBL.lrDispencer1DoseValveOpenVolumeShow.lrValue    									:=						STRING_TO_LREAL (aRecipeParamsValues[61 ]);
stActRecipe.stUBL.lrDispencer1DoseValveOpenTimeAccShow.lrValue   									:=						STRING_TO_LREAL (aRecipeParamsValues[62 ]);
stActRecipe.stUBL.lrDispencer1DoseValveCloseVolumeShow.lrValue    									:=						STRING_TO_LREAL (aRecipeParamsValues[63 ]);
stActRecipe.stUBL.lrDispencer1DoseValveCloseTimeDecShow.lrValue 									:=						STRING_TO_LREAL (aRecipeParamsValues[64 ]);
stActRecipe.stUBL.lrDispencer1DoseSuckingVolumeShow.lrValue 										:=						STRING_TO_LREAL (aRecipeParamsValues[65 ]);
stActRecipe.stUBL.lrDispencer1DoseSuckingTimeDelayShow.lrValue 										:=						STRING_TO_LREAL (aRecipeParamsValues[66 ]);
stActRecipe.stUBL.bDispencer1DoseSuckingShow.bValue 			       								:=						STRING_TO_BOOL	(aRecipeParamsValues[67 ]);
stActRecipe.stUBL.bDispencer1LiftSynchroPh1Show.bValue 												:=						STRING_TO_BOOL	(aRecipeParamsValues[68 ]);
stActRecipe.stUBL.bDispencer1LiftSynchroPh2Show.bValue 			   									:=						STRING_TO_BOOL	(aRecipeParamsValues[69 ]);
stActRecipe.stUBL.bDispencer1LiftSynchroPh3Show.bValue 		       									:=						STRING_TO_BOOL	(aRecipeParamsValues[70 ]);
stActRecipe.stUBL.lrDispencer1LifterStartDosePositionShow.lrValue									:=						STRING_TO_LREAL (aRecipeParamsValues[71 ]);
stActRecipe.stUBL.lrDispencer1LifterStopDosePositionShow.lrValue 									:=						STRING_TO_LREAL (aRecipeParamsValues[72 ]);
stActRecipe.stUBL.lrDispencer1LifterVelocityShow.lrValue            								:=						STRING_TO_LREAL (aRecipeParamsValues[73 ]);
stActRecipe.stUBL.lrDispencer1LifterAccelerationShow.lrValue        								:=						STRING_TO_LREAL (aRecipeParamsValues[74 ]);
stActRecipe.stUBL.lrDispencer1LifterDecelerationShow.lrValue 		    							:=						STRING_TO_LREAL (aRecipeParamsValues[75 ]);
stActRecipe.stUBL.lrDispencer2DoseVolumeShow.lrValue	            								:=						STRING_TO_LREAL (aRecipeParamsValues[76 ]);
stActRecipe.stUBL.lrDispencer2Phase1VolumeShow.lrValue 			    								:=						STRING_TO_LREAL (aRecipeParamsValues[77 ]);
stActRecipe.stUBL.lrDispencer2Phase2VolumeShow.lrValue 			    								:=						STRING_TO_LREAL (aRecipeParamsValues[78 ]);
stActRecipe.stUBL.lrDispencer2Phase1VelocityShow.lrValue 		    								:=						STRING_TO_LREAL (aRecipeParamsValues[79 ]);
stActRecipe.stUBL.lrDispencer2Phase2VelocityShow.lrvalue 		    								:=						STRING_TO_LREAL (aRecipeParamsValues[80 ]);
stActRecipe.stUBL.lrDispencer2Phase3VelocityShow.lrValue 		    								:=						STRING_TO_LREAL (aRecipeParamsValues[81 ]);
stActRecipe.stUBL.lrDispencer2SuckVelocityShow.lrValue     											:=						STRING_TO_LREAL (aRecipeParamsValues[82 ]);
stActRecipe.stUBL.lrDispencer2Phase1AccelerationShow.lrValue 	        							:=						STRING_TO_LREAL (aRecipeParamsValues[83 ]);
stActRecipe.stUBL.lrDispencer2Phase2AccelerationShow.lrValue 	        							:=						STRING_TO_LREAL (aRecipeParamsValues[84 ]);
stActRecipe.stUBL.lrDispencer2Phase3AccelerationShow.lrValue 		    							:=						STRING_TO_LREAL (aRecipeParamsValues[85 ]);
stActRecipe.stUBL.lrDispencer2SuckAccelerationShow.lrValue   										:=						STRING_TO_LREAL (aRecipeParamsValues[86 ]);
stActRecipe.stUBL.lrDispencer2Phase1DecelerationShow.lrValue 										:=						STRING_TO_LREAL (aRecipeParamsValues[87 ]);
stActRecipe.stUBL.lrDispencer2Phase2DecelerationShow.lrValue 										:=						STRING_TO_LREAL (aRecipeParamsValues[88 ]);
stActRecipe.stUBL.lrDispencer2Phase3DecelerationShow.lrValue 										:=						STRING_TO_LREAL (aRecipeParamsValues[89 ]);
stActRecipe.stUBL.udiDispencer2DosingDoneDelayTimeShow.udiValue 									:=						STRING_TO_UDINT (aRecipeParamsValues[90 ]);
stActRecipe.stUBL.lrDispencer2SuckValveOpenVolumeShow.lrValue 										:=						STRING_TO_LREAL (aRecipeParamsValues[91 ]);
stActRecipe.stUBL.lrDispencer2SuckValveOpenTimeDelayShow.lrValue 									:=						STRING_TO_LREAL (aRecipeParamsValues[92 ]);
stActRecipe.stUBL.lrDispencer2SuckValveCloseVolumeShow.lrValue										:=						STRING_TO_LREAL (aRecipeParamsValues[93 ]);
stActRecipe.stUBL.lrDispencer2SuckValveCloseTimeDelayShow.lrValue 									:=						STRING_TO_LREAL (aRecipeParamsValues[94 ]);
stActRecipe.stUBL.lrDispencer2DoseValveOpenVolumeShow.lrValue 										:=						STRING_TO_LREAL (aRecipeParamsValues[95 ]);
stActRecipe.stUBL.lrDispencer2DoseValveOpenTimeAccShow.lrValue 										:=						STRING_TO_LREAL (aRecipeParamsValues[96 ]);
stActRecipe.stUBL.lrDispencer2DoseValveCloseVolumeShow.lrValue 										:=						STRING_TO_LREAL (aRecipeParamsValues[97 ]);
stActRecipe.stUBL.lrDispencer2DoseValveCloseTimeDecShow.lrValue										:=						STRING_TO_LREAL (aRecipeParamsValues[98 ]);
stActRecipe.stUBL.lrDispencer2DoseSuckingVolumeShow.lrValue	    									:=						STRING_TO_LREAL (aRecipeParamsValues[99 ]);
stActRecipe.stUBL.lrDispencer2DoseSuckingTimeDelayShow.lrValue										:=						STRING_TO_LREAL (aRecipeParamsValues[100]);
stActRecipe.stUBL.bDispencer2DoseSuckingShow.bValue 	            								:=						STRING_TO_BOOL	(aRecipeParamsValues[101]);
stActRecipe.stUBL.bDispencer2LiftSynchroPh1Show.bValue 	        									:=						STRING_TO_BOOL	(aRecipeParamsValues[102]);
stActRecipe.stUBL.bDispencer2LiftSynchroPh2Show.bValue 	        									:=						STRING_TO_BOOL	(aRecipeParamsValues[103]);
stActRecipe.stUBL.bDispencer2LiftSynchroPh3Show.bValue 	        									:=						STRING_TO_BOOL	(aRecipeParamsValues[104]);
stActRecipe.stUBL.lrDispencer2LifterStartDosePositionShow.lrValue									:=						STRING_TO_LREAL (aRecipeParamsValues[105]);
stActRecipe.stUBL.lrDispencer2LifterStopDosePositionShow.lrValue 									:=						STRING_TO_LREAL (aRecipeParamsValues[106]);
stActRecipe.stUBL.lrDispencer2LifterVelocityShow.lrValue        									:=						STRING_TO_LREAL (aRecipeParamsValues[107]);
stActRecipe.stUBL.lrDispencer2LifterAccelerationShow.lrValue 										:=						STRING_TO_LREAL (aRecipeParamsValues[108]);
stActRecipe.stUBL.lrDispencer2LifterDecelerationShow.lrValue 	    								:=						STRING_TO_LREAL (aRecipeParamsValues[109]);
stActRecipe.stUBL.bDispencersCatchEnableShow.bValue             									:=				   		STRING_TO_BOOL	(aRecipeParamsValues[110]); 	
stActRecipe.stUBL.bDispencersCatchMaxPressureShow.bValue          									:=			   			STRING_TO_BOOL	(aRecipeParamsValues[111]);
stActRecipe.stUBL.lrDispencersCatchHeightSVShow.lrValue												:=						STRING_TO_LREAL (aRecipeParamsValues[112]);	
stActRecipe.stUBL.lrDispencersCatch1ClosedValueShow.lrValue          								:=						STRING_TO_LREAL (aRecipeParamsValues[113]);	
stActRecipe.stUBL.lrDispencersCatch1OpenValueShow.lrValue          									:=						STRING_TO_LREAL (aRecipeParamsValues[114]); 
stActRecipe.stUBL.lrDispencersCatch2ClosedValueShow.lrValue       									:=						STRING_TO_LREAL (aRecipeParamsValues[115]); 
stActRecipe.stUBL.lrDispencersCatch2OpenValueShow.lrValue	    									:=						STRING_TO_LREAL (aRecipeParamsValues[116]);	
stActRecipe.stUBL.lrDispencersCatch3ClosedValueShow.lrValue         								:=						STRING_TO_LREAL (aRecipeParamsValues[117]);
stActRecipe.stUBL.lrDispencersCatch3OpenValueShow.lrValue           								:=						STRING_TO_LREAL (aRecipeParamsValues[118]);	
stActRecipe.stUBL.lrDispencersCatch4ClosedValueShow.lrValue         								:=						STRING_TO_LREAL (aRecipeParamsValues[119]);	
stActRecipe.stUBL.lrDispencersCatch4OpenValueShow.lrValue											:=						STRING_TO_LREAL (aRecipeParamsValues[120]); 
stActRecipe.stUBL.lrDispencersCatchToleranceShow.lrValue 	        								:=						STRING_TO_LREAL (aRecipeParamsValues[121]); 	
stActRecipe.stUBL.bTank1MixerEnableShow.bValue    													:=						STRING_TO_BOOL	(aRecipeParamsValues[122]);
stActRecipe.stUBL.bTankHeatingEnableShow.bValue   													:=						STRING_TO_BOOL	(aRecipeParamsValues[123]);
stActRecipe.stUBL.iTankHeatingTempSVShow.diValue  													:=				        STRING_TO_DINT  (aRecipeParamsValues[124]);
stActRecipe.stUBL.bTank1PressureEnableShow.bValue													:=				        STRING_TO_BOOL  (aRecipeParamsValues[125]);
stActRecipe.stUBL.bTank1SupplyPumpEnableShow.bValue                             					:=                      STRING_TO_BOOL  (aRecipeParamsValues[126]);
stActRecipe.stUBL.bTank2SupplyPumpEnableShow.bValue                             					:=                      STRING_TO_BOOL  (aRecipeParamsValues[127]);
stActRecipe.stUBL.uTank1LevelSetpointShow.udiValue                              					:=                      STRING_TO_UDINT (aRecipeParamsValues[128]);
stActRecipe.stUBL.uTank2LevelSetpointShow.udiValue                              					:=                      STRING_TO_UDINT (aRecipeParamsValues[129]);
stActRecipe.stUBL.bTank1LevelSignalInvertShow.bValue 	                        					:=                      STRING_TO_BOOL  (aRecipeParamsValues[130]);
stActRecipe.stUBL.bTank2LevelSignalInvertShow.bValue 	                        					:=                      STRING_TO_BOOL  (aRecipeParamsValues[131]);
stActRecipe.stUBL.bWeight1EnableShow.bValue                                     					:=       				STRING_TO_BOOL  (aRecipeParamsValues[132]);
stActRecipe.stUBL.lrWeightMassSVShow.lrValue	                                					:=       				STRING_TO_LREAL (aRecipeParamsValues[133]);
stActRecipe.stUBL.iWeight1ActuatorUpDelayShow.diValue 												:=			            STRING_TO_DINT  (aRecipeParamsValues[134]);
stActRecipe.stUBL.iWeight2ActuatorUpDelayShow.diValue                           					:=                      STRING_TO_DINT  (aRecipeParamsValues[135]);
stActRecipe.stUBL.iWeight3ActuatorUpDelayShow.diValue                           					:=                      STRING_TO_DINT  (aRecipeParamsValues[136]);
stActRecipe.stUBL.iWeight4ActuatorUpDelayShow.diValue                           					:=                      STRING_TO_DINT  (aRecipeParamsValues[137]);
stActRecipe.stUBL.iWeight5ActuatorUpDelayShow.diValue                           					:=                      STRING_TO_DINT  (aRecipeParamsValues[138]);
stActRecipe.stUBL.iWeight6ActuatorUpDelayShow.diValue                           					:=                      STRING_TO_DINT  (aRecipeParamsValues[139]);
stActRecipe.stUBL.lrFormWeightShow.lrValue                                      					:=						STRING_TO_LREAL (aRecipeParamsValues[140]);
stActRecipe.stUBL.lrMass1DensityShow.lrValue                                    					:=						STRING_TO_LREAL (aRecipeParamsValues[141]);
stActRecipe.stUBL.lrMass2DensityShow.lrValue                                    					:=						STRING_TO_LREAL (aRecipeParamsValues[142]);
stActRecipe.stUBL.lrCupWeightShow.lrValue                                       					:=						STRING_TO_LREAL (aRecipeParamsValues[143]);
stActRecipe.stUBL.lrWholePackageWeightShow.lrValue 	                            					:=					    STRING_TO_LREAL (aRecipeParamsValues[144]);
stActRecipe.stUBL.lrWeight1MeasurmentCorrectionShow.lrValue	                    					:=					    STRING_TO_LREAL (aRecipeParamsValues[145]);
stActRecipe.stUBL.bDispencer1WeightCorrectionEnableShow.bValue                  					:=					    STRING_TO_BOOL  (aRecipeParamsValues[146]);
stActRecipe.stUBL.bDispencer2WeightCorrectionEnableShow.bValue                  					:=					    STRING_TO_BOOL  (aRecipeParamsValues[147]);
stActRecipe.stUBL.bDispencer3WeightCorrectionEnableShow.bValue                  					:=					    STRING_TO_BOOL  (aRecipeParamsValues[148]);
stActRecipe.stUBL.bDispencer4WeightCorrectionEnableShow.bValue                  					:=					    STRING_TO_BOOL  (aRecipeParamsValues[149]);
stActRecipe.stUBL.lrWeightUpperToleranceShow.lrValue                            					:=					    STRING_TO_LREAL (aRecipeParamsValues[150]);
stActRecipe.stUBL.lrWeightLowerToleranceShow.lrValue                            					:=					    STRING_TO_LREAL (aRecipeParamsValues[151]);
stActRecipe.stUBL.iWeightCorrectionNumberOfSamplesShow.udiValue                 					:=					    STRING_TO_UDINT (aRecipeParamsValues[152]);
stActRecipe.stUBL.bLidFeederEnableShow.bValue                 										:=						STRING_TO_BOOL  (aRecipeParamsValues[153]);
stActRecipe.stUBL.bLidFeederHeaterEnableShow.bValue                             					:=					    STRING_TO_BOOL  (aRecipeParamsValues[154]);
stActRecipe.stUBL.lrLidFeederHeightPosSVShow.lrValue                            					:=					    STRING_TO_LREAL (aRecipeParamsValues[155]);
stActRecipe.stUBL.iLidFeederHeatingTimeShow.diValue                             					:=					    STRING_TO_DINT  (aRecipeParamsValues[156]);
stActRecipe.stUBL.iLidFeederTempHisteresisShow.diValue                          					:=					    STRING_TO_DINT  (aRecipeParamsValues[157]);
stActRecipe.stUBL.iLidFeeder1TempSVShow.diValue 	                            					:=					    STRING_TO_DINT  (aRecipeParamsValues[158]);
stActRecipe.stUBL.iLidFeeder2TempSVShow.diValue 	                            					:=					    STRING_TO_DINT  (aRecipeParamsValues[159]);
stActRecipe.stUBL.bLidFeederDragingStationEnableShow.bValue 	                					:=                      STRING_TO_BOOL  (aRecipeParamsValues[160]);
stActRecipe.stUBL.lrLidFeederDragingStationVelocityShow.lrValue	                					:=                      STRING_TO_LREAL (aRecipeParamsValues[161]);
stActRecipe.stUBL.lrLidFeederDragingStationAccelerationShow.lrValue	            					:=                      STRING_TO_LREAL (aRecipeParamsValues[162]);
stActRecipe.stUBL.lrLidFeederDragingStationDecelerationShow.lrValue	            					:=                      STRING_TO_LREAL (aRecipeParamsValues[163]);
stActRecipe.stUBL.bLidPuttedCheckEnableShow.bValue                              					:=                      STRING_TO_BOOL  (aRecipeParamsValues[164]);
stActRecipe.stUBL.lrLidPuttedCheckHeightSVShow.lrValue                          					:=                      STRING_TO_LREAL (aRecipeParamsValues[165]);
stActRecipe.stUBL.lrLidPuttedCheckPositionShow.lrValue                          					:=                      STRING_TO_LREAL (aRecipeParamsValues[166]);
stActRecipe.stUBL.lrLidPuttedCheckAreaShow.lrValue                              					:=                      STRING_TO_LREAL (aRecipeParamsValues[167]);
stActRecipe.stUBL.iLidPuttedCheckProgramShow.diValue                            					:=      				STRING_TO_DINT  (aRecipeParamsValues[168]);
stActRecipe.stUBL.bLidSealerEnableShow.bValue                                   					:=      				STRING_TO_BOOL  (aRecipeParamsValues[169]);
stActRecipe.stUBL.bLidSealerHeaterEnableShow.bValue 	                        					:=      				STRING_TO_BOOL  (aRecipeParamsValues[170]);
stActRecipe.stUBL.iLidSealerHeatingTimeShow.diValue	                            					:=      				STRING_TO_DINT  (aRecipeParamsValues[171]);
stActRecipe.stUBL.lrLidSealerPressureShow.lrValue                               					:=      				STRING_TO_LREAL (aRecipeParamsValues[172]);
stActRecipe.stUBL.lrLidSealerHeightPosSVShow.lrValue                            					:=      				STRING_TO_LREAL (aRecipeParamsValues[173]);
stActRecipe.stUBL.iLidSealerTempHisteresisShow.diValue                          					:=      				STRING_TO_DINT  (aRecipeParamsValues[174]);
stActRecipe.stUBL.iLidSealer1TempSVShow.diValue 	                            					:=      				STRING_TO_DINT  (aRecipeParamsValues[175]);
stActRecipe.stUBL.iLidSealer2TempSVShow.diValue 	                            					:=      				STRING_TO_DINT  (aRecipeParamsValues[176]);
stActRecipe.stUBL.bLidSealerDragingStationEnableShow.bValue                     					:=      		        STRING_TO_BOOL  (aRecipeParamsValues[177]);
stActRecipe.stUBL.lrLidSealerDragingStationVelocityShow.lrValue 	            					:=      				STRING_TO_LREAL (aRecipeParamsValues[178]);
stActRecipe.stUBL.lrLidSealerDragingStationAccelerationShow.lrValue	            					:=      				STRING_TO_LREAL (aRecipeParamsValues[179]);
stActRecipe.stUBL.lrLidSealerDragingStationDecelerationShow.lrValue	            					:=      				STRING_TO_LREAL (aRecipeParamsValues[180]);
stActRecipe.stUBL.bCapFeederGateEnableShow.bValue 	                            					:=      				STRING_TO_BOOL  (aRecipeParamsValues[181]);
stActRecipe.stUBL.iCapFeederGateBlockingTimeShow.diValue 	                    					:=      				STRING_TO_DINT  (aRecipeParamsValues[182]);
stActRecipe.stUBL.bCapFeederEnableShow.bValue                                   					:=      				STRING_TO_BOOL  (aRecipeParamsValues[183]);
stActRecipe.stUBL.lrCapFeederHeightPosSVShow.lrValue                            					:=                      STRING_TO_LREAL (aRecipeParamsValues[184]);
stActRecipe.stUBL.iCapFeederTimeDelayOnShow.diValue                             					:=                      STRING_TO_DINT  (aRecipeParamsValues[185]);
stActRecipe.stUBL.iCapFeederTimeDelayOffShow.diValue                            					:=                      STRING_TO_DINT  (aRecipeParamsValues[186]);
stActRecipe.stUBL.iCapFeederTimeToEmptySleeveErrorShow.diValue                  					:=                      STRING_TO_DINT  (aRecipeParamsValues[187]);
stActRecipe.stUBL.bCapSorterOnlyWeightOKEnableShow.bValue                       					:=                      STRING_TO_BOOL  (aRecipeParamsValues[188]);
stActRecipe.stUBL.bCapSorterDragEnableShow.bValue                               					:=                      STRING_TO_BOOL  (aRecipeParamsValues[189]);
stActRecipe.stUBL.lrCapSorterDragVelocityShow.lrValue                           					:=                      STRING_TO_LREAL (aRecipeParamsValues[190]);
stActRecipe.stUBL.lrCapSorterDragAccelerationShow.lrValue 	                    					:=                      STRING_TO_LREAL (aRecipeParamsValues[191]);
stActRecipe.stUBL.lrCapSorterDragDecelerationShow.lrValue 	                    					:=                      STRING_TO_LREAL (aRecipeParamsValues[192]);
stActRecipe.stUBL.bCapPuttedCheckEnableShow.bValue                              					:=                      STRING_TO_BOOL  (aRecipeParamsValues[193]);
stActRecipe.stUBL.lrCapPuttedCheckHeightPosSVShow.lrValue 	                    					:=                      STRING_TO_LREAL (aRecipeParamsValues[194]);
stActRecipe.stUBL.bGripperScrewer1EnableShow.bValue 	                        					:=                      STRING_TO_BOOL  (aRecipeParamsValues[195]);
stActRecipe.stUBL.lrGripperScrewingTightTorqueShow.lrValue                      					:=                      STRING_TO_LREAL (aRecipeParamsValues[196]);
stActRecipe.stUBL.bGripperScrewer2EnableShow.bValue 	                        					:=                      STRING_TO_BOOL  (aRecipeParamsValues[197]);
stActRecipe.stUBL.lrGripperScrewing2TightTorqueShow.lrValue	                    					:=                      STRING_TO_LREAL (aRecipeParamsValues[198]);
stActRecipe.stUBL.iGripperScrewer1ToolShow.diValue                              					:=                      STRING_TO_DINT  (aRecipeParamsValues[199]);
stActRecipe.stUBL.lrGripperScrewer1VelocityShow.lrValue                         					:=                      STRING_TO_LREAL (aRecipeParamsValues[200]);
stActRecipe.stUBL.nGripperScrewer1TightTimeShow.diValue	                        					:=                      STRING_TO_DINT  (aRecipeParamsValues[201]);
stActRecipe.stUBL.iGripperScrewer1StartDelayShow.diValue	                    					:=                      STRING_TO_DINT  (aRecipeParamsValues[202]);
stActRecipe.stUBL.lrGripperScrewerReadyPositionShow.lrValue 	                					:=                      STRING_TO_LREAL (aRecipeParamsValues[203]);
stActRecipe.stUBL.lrGripperScrewerPushingCapPositionShow.lrValue 	            					:=                      STRING_TO_LREAL (aRecipeParamsValues[204]);
stActRecipe.stUBL.lrGripperScrewerScrewingCapPositionShow.lrValue               					:=                      STRING_TO_LREAL (aRecipeParamsValues[205]);
stActRecipe.stUBL.lrGripperScrewerPressureShow.lrValue                          					:=                      STRING_TO_LREAL (aRecipeParamsValues[206]);
stActRecipe.stUBL.lrGripperScrewerCatchPressureShow.lrValue 	                					:=                      STRING_TO_LREAL (aRecipeParamsValues[207]);
stActRecipe.stUBL.lrDispencerCatchPressureShow.lrValue                          					:=                      STRING_TO_LREAL (aRecipeParamsValues[208]);
stActRecipe.stUBL.lrGripperScrewerPressureExhaustLevelShow.lrValue              					:=                      STRING_TO_LREAL (aRecipeParamsValues[209]);
stActRecipe.stUBL.lrGripperScrewerCatchPressureExhaustLevelShow.lrValue         					:=                      STRING_TO_LREAL (aRecipeParamsValues[210]);
stActRecipe.stUBL.lrGripperScrewerTurnoversToFullScrewedShow.lrValue 	        					:=                      STRING_TO_LREAL (aRecipeParamsValues[211]);
stActRecipe.stUBL.lrGripperScrewerThreadPitchShow.lrValue                       					:=                      STRING_TO_LREAL (aRecipeParamsValues[212]);
stActRecipe.stUBL.lrGripperScrewerThreadTimesShow.lrValue                       					:=                      STRING_TO_LREAL (aRecipeParamsValues[213]);
stActRecipe.stUBL.nGripperScrewerCatchHeightSVShow.diValue	                    					:=       			    STRING_TO_DINT  (aRecipeParamsValues[214]);
stActRecipe.stUBL.bGripperScrewer1FindScrewShow.bValue                          					:=      			    STRING_TO_BOOL  (aRecipeParamsValues[215]);
stActRecipe.stUBL.bGripperScrewer1Option4Show.bValue                            					:=    			        STRING_TO_BOOL  (aRecipeParamsValues[216]);
stActRecipe.stUBL.lrGripperScrewer1FindingScrewDegreeShow.lrValue               					:=    			        STRING_TO_LREAL (aRecipeParamsValues[217]);
stActRecipe.stUBL.bGripperScrewer1Option1Show.bValue	                        					:=       			    STRING_TO_BOOL  (aRecipeParamsValues[218]);
stActRecipe.stUBL.bGripperScrewer1Option2Show.bValue	                        					:=       			    STRING_TO_BOOL  (aRecipeParamsValues[219]);
stActRecipe.stUBL.bGripperScrewer1Option3Show.bValue	                        					:=       			    STRING_TO_BOOL  (aRecipeParamsValues[220]);
stActRecipe.stUBL.bGripperScrewer1Option5Show.bValue	                        					:=       			    STRING_TO_BOOL  (aRecipeParamsValues[221]);
stActRecipe.stUBL.bGripperScrewer1Option6Show.bValue	                        					:=       			    STRING_TO_BOOL  (aRecipeParamsValues[222]);
stActRecipe.stUBL.bGripperScrewer1Option7Show.bValue	                        					:=       			    STRING_TO_BOOL  (aRecipeParamsValues[223]);
stActRecipe.stUBL.bBottleDragingStationEnableShow.bValue 	                    					:=       			    STRING_TO_BOOL  (aRecipeParamsValues[224]);
stActRecipe.stUBL.lrBottleDragingStationVelocityShow.lrValue                    					:=    			        STRING_TO_LREAL (aRecipeParamsValues[225]);
stActRecipe.stUBL.bCapCorrectCheckEnableShow.bValue 	                        					:=       		        STRING_TO_BOOL  (aRecipeParamsValues[226]);
stActRecipe.stUBL.lrCapCorrectCheckHeightPosSVShow.lrValue                      					:=      			    STRING_TO_LREAL (aRecipeParamsValues[227]);
stActRecipe.stUBL.bCapCorrectCheckCameraEnableShow.bValue                       					:=     			        STRING_TO_BOOL  (aRecipeParamsValues[228]);
stActRecipe.stUBL.iCapCorrectCheckCameraProgramShow.diValue 	                					:=           			STRING_TO_DINT  (aRecipeParamsValues[229]);
stActRecipe.stUBL.bBottleTransferEnableShow.bValue			                    					:=       			    STRING_TO_BOOL  (aRecipeParamsValues[230]);
stActRecipe.stUBL.nBottleTransferProgramShow.udiValue			                					:=           		    STRING_TO_UDINT (aRecipeParamsValues[231]);
stActRecipe.stUBL.iBottleTransferPickOffsetXShow.diValue                        					:=     			        STRING_TO_DINT  (aRecipeParamsValues[232]);
stActRecipe.stUBL.iBottleTransferPickOffsetYShow.diValue 	                    					:=       			    STRING_TO_DINT  (aRecipeParamsValues[233]);
stActRecipe.stUBL.iBottleTransferPickOffsetZShow.diValue                        					:=     			        STRING_TO_DINT  (aRecipeParamsValues[234]);
stActRecipe.stUBL.iBottleTransferPick2OffsetXShow.diValue                       					:=     			        STRING_TO_DINT  (aRecipeParamsValues[235]);
stActRecipe.stUBL.iBottleTransferPick2OffsetYShow.diValue 	                    					:=       			    STRING_TO_DINT  (aRecipeParamsValues[236]);
stActRecipe.stUBL.iBottleTransferPick2OffsetZShow.diValue                       					:=    			        STRING_TO_DINT  (aRecipeParamsValues[237]);
stActRecipe.stUBL.iBottleTransferPlace1OffsetXShow.diValue 	                    					:=       			    STRING_TO_DINT  (aRecipeParamsValues[238]);
stActRecipe.stUBL.iBottleTransferPlace1OffsetYShow.diValue 	                    					:=       			    STRING_TO_DINT  (aRecipeParamsValues[239]);
stActRecipe.stUBL.iBottleTransferPlace1OffsetZShow.diValue 	                    					:=       			    STRING_TO_DINT  (aRecipeParamsValues[240]);
stActRecipe.stUBL.iBottleTransferPlace2OffsetXShow.diValue 	                    					:=       			    STRING_TO_DINT  (aRecipeParamsValues[241]);
stActRecipe.stUBL.iBottleTransferPlace2OffsetYShow.diValue 	                    					:=       			    STRING_TO_DINT  (aRecipeParamsValues[242]);
stActRecipe.stUBL.iBottleTransferPlace2OffsetZShow.diValue 	                    					:=       			    STRING_TO_DINT  (aRecipeParamsValues[243]);
stActRecipe.stUBL.iBottleTransferSpeedShow.diValue 	                            					:=       			    STRING_TO_DINT  (aRecipeParamsValues[244]);
stActRecipe.stUBL.bBottleTransferInkJetEnableShow.bValue 	                    					:=       			    STRING_TO_BOOL  (aRecipeParamsValues[245]);
stActRecipe.stUBL.bBottleTransferPickOnlyOneShow.bValue                         					:=   				    STRING_TO_BOOL  (aRecipeParamsValues[246]);
stActRecipe.stUBL.bBottleTransferWeightEnableShow.bValue 	                    					:=       			    STRING_TO_BOOL  (aRecipeParamsValues[247]);
stActRecipe.stUBL.iBottleTransferWeightIntervalShow.diValue	                    					:=         		        STRING_TO_DINT  (aRecipeParamsValues[248]);
stActRecipe.stUBL.bBottleTransferRotateEnableShow.bValue 	                    					:=         		        STRING_TO_BOOL  (aRecipeParamsValues[249]);
stActRecipe.stUBL.bBadBottleConveyorEnableShow.bValue                           					:=       		        STRING_TO_BOOL  (aRecipeParamsValues[250]);
stActRecipe.stUBL.nBadBottleConveyorVelocitySVShow.udiValue 	                					:=             		    STRING_TO_UDINT (aRecipeParamsValues[251]);
stActRecipe.stUBL.bLabelMachineEnableShow.bValue 	                            					:=         		        STRING_TO_BOOL  (aRecipeParamsValues[252]);
stActRecipe.stUBL.bExitTurnTable1EnableShow.bValue                              					:=       		        STRING_TO_BOOL  (aRecipeParamsValues[253]);
stActRecipe.stUBL.bExitConveyorEnableShow.bValue                                					:=     		            STRING_TO_BOOL  (aRecipeParamsValues[254]);
stActRecipe.stUBL.nExitConveyorVelocitySVShow.udiValue 	                        					:=         		        STRING_TO_UDINT (aRecipeParamsValues[255]);
stActRecipe.stUBL.bFormTransportersEnableShow.bValue						    					:=         			    STRING_TO_BOOL  (aRecipeParamsValues[256]);
stActRecipe.stUBL.nFormTransportersDispencerVelocitySVShow.udiValue	            					:=      		        STRING_TO_UDINT (aRecipeParamsValues[257]);
stActRecipe.stUBL.nFormTransportersScrewerVelocitySVShow.udiValue			    					:=             	        STRING_TO_UDINT (aRecipeParamsValues[258]);
stActRecipe.stUBL.nFormTransportersBeforeScrewerVelocitySVShow.udiValue	        					:=         		        STRING_TO_UDINT (aRecipeParamsValues[259]);
stActRecipe.stUBL.nFormTransportersSlowerVelocitySVShow.udiValue		 	    					:=             		    STRING_TO_UDINT (aRecipeParamsValues[260]);
stActRecipe.stUBL.bCircularInkjetEnableShow.bValue	 	                        					:=         		        STRING_TO_BOOL  (aRecipeParamsValues[261]);
stActRecipe.stUBL.iCircularInkjetSpeedShow.diValue	 	                        					:=         		        STRING_TO_DINT  (aRecipeParamsValues[262]);
stActRecipe.stUBL.iCircularInkjetDelayShow.diValue	 	                        					:=         		        STRING_TO_DINT  (aRecipeParamsValues[263]);
stActRecipe.stUBL.iCircularInkjetHoldShow.diValue	 	                        					:=         		        STRING_TO_DINT  (aRecipeParamsValues[264]);
stActRecipe.stUCF.iCapSorterProductType.diValue 	                            					:=             		    STRING_TO_DINT  (aRecipeParamsValues[265]);
stActRecipe.stUCF.uiCapSorterIndexShow.udiValue 													:=				        STRING_TO_UDINT (aRecipeParamsValues[266]);
stActRecipe.stUCF.bPresenceBottleEnableShow.bValue 	                            					:=         		        STRING_TO_BOOL  (aRecipeParamsValues[267]);
stActRecipe.stUCF.bCapSorterTransporterEnableShow.bValue											:=			  		    STRING_TO_BOOL  (aRecipeParamsValues[268]);
stActRecipe.stUCF.iCapSorterTransporterTankConveyorVelocityShow.diValue								:=	 	                STRING_TO_DINT  (aRecipeParamsValues[269]);
stActRecipe.stUCF.iCapSorterTransporterStartDelayTimeShow.diValue									:=		                STRING_TO_DINT  (aRecipeParamsValues[270]);
stActRecipe.stUCF.udiCapSorterTransporterTimeProductOnSensorBeforeBrushShow.udiValue				:=			            STRING_TO_UDINT (aRecipeParamsValues[271]);
stActRecipe.stUCF.iCapSorterTransporterEmptyingConveyorSpeedShow.diValue							:=				        STRING_TO_DINT  (aRecipeParamsValues[272]);
stActRecipe.stUCF.iCapSorterTransporterVolumeOfCapsShow.diValue										:=	 	                STRING_TO_DINT  (aRecipeParamsValues[273]);
stActRecipe.stUCF.bCapSorterWheelEnableShow.bValue							    					:=  		            STRING_TO_BOOL  (aRecipeParamsValues[274]);
stActRecipe.stUCF.lrCapSorterWheelMoveAccelerationEmptyTableShow.lrValue	    					:=    		            STRING_TO_LREAL (aRecipeParamsValues[275]);
stActRecipe.stUCF.lrCapSorterWheelMoveDecelerationEmptyTableShow.lrValue	    					:=    		            STRING_TO_LREAL (aRecipeParamsValues[276]);
stActRecipe.stUCF.lrCapSorterWheelMoveSpeedEmptyTableShow.lrValue			    					:=		                STRING_TO_LREAL (aRecipeParamsValues[277]);
stActRecipe.stUCF.lrCapSorterWheelMoveAngleEmptyTableShow.lrValue			    					:=		                STRING_TO_LREAL (aRecipeParamsValues[278]);
stActRecipe.stUCF.lrCapSorterWheelJerkAngleEmptyTableShow.lrValue			    					:=		                STRING_TO_LREAL (aRecipeParamsValues[279]);
stActRecipe.stUCF.iCapSorterWheelWaitingAfterRotationEmptyTableShow.diValue     					:=      		        STRING_TO_DINT  (aRecipeParamsValues[280]);
stActRecipe.stUCF.lrCapSorterWheelMoveAccelerationFullTableShow.lrValue	        					:=  		            STRING_TO_LREAL (aRecipeParamsValues[281]);
stActRecipe.stUCF.lrCapSorterWheelMoveDecelerationFullTableShow.lrValue	        					:=  		            STRING_TO_LREAL (aRecipeParamsValues[282]);
stActRecipe.stUCF.lrCapSorterWheelMoveSpeedFullTableShow.lrValue			    					:=        		        STRING_TO_LREAL (aRecipeParamsValues[283]);
stActRecipe.stUCF.lrCapSorterWheelMoveAngleFullyTableShow.lrValue			    					:=     		            STRING_TO_LREAL (aRecipeParamsValues[284]);
stActRecipe.stUCF.lrCapSorterWheelJerkAngleFullTableShow.lrValue			    					:=      		        STRING_TO_LREAL (aRecipeParamsValues[285]);
stActRecipe.stUCF.iCapSorterWheelWaitingAfterRotationFullTableShow.diValue      					:= 			            STRING_TO_DINT  (aRecipeParamsValues[286]);
stActRecipe.stUCF.lrCapSorterWheelMoveAccelerationHalfFullTableShow.lrValue     					:= 			            STRING_TO_LREAL (aRecipeParamsValues[287]);
stActRecipe.stUCF.lrCapSorterWheelMoveDecelerationHalfFullTableShow.lrValue     					:= 			            STRING_TO_LREAL (aRecipeParamsValues[288]);
stActRecipe.stUCF.lrCapSorterWheelMoveSpeedHalfFullTableShow.lrValue								:=       			    STRING_TO_LREAL (aRecipeParamsValues[289]);
stActRecipe.stUCF.lrCapSorterWheelMoveAngleHalfFullyTableShow.lrValue								:=   			        STRING_TO_LREAL (aRecipeParamsValues[290]);
stActRecipe.stUCF.lrCapSorterWheelJerkAngleHalfFullTableShow.lrValue								:=       			    STRING_TO_LREAL (aRecipeParamsValues[291]);
stActRecipe.stUCF.iCapSorterWheelWaitingAfterRotationHalfFullTableShow.diValue 						:=       			    STRING_TO_DINT  (aRecipeParamsValues[292]);
stActRecipe.stUCF.bCapSorterCameraEnableShow.bValue                            						:=		                STRING_TO_BOOL  (aRecipeParamsValues[293]);
stActRecipe.stUCF.bCapSorterRobotEnableShow.bValue                 			    					:=                      STRING_TO_BOOL  (aRecipeParamsValues[294]);
stActRecipe.stUCF.lrCapSorterRobotPlace1PositionXShow.lrValue										:=		                STRING_TO_LREAL (aRecipeParamsValues[295]);
stActRecipe.stUCF.lrCapSorterRobotPlace1PositionYShow.lrValue										:=		                STRING_TO_LREAL (aRecipeParamsValues[296]);
stActRecipe.stUCF.lrCapSorterRobotPlace1PositionZShow.lrValue										:=		                STRING_TO_LREAL (aRecipeParamsValues[297]);
stActRecipe.stUCF.lrCapSorterRobotPlace1PositionCShow.lrValue										:=		                STRING_TO_LREAL (aRecipeParamsValues[298]);
stActRecipe.stUCF.iCapSorterRobotPickElevationShow.diValue											:=		                STRING_TO_DINT  (aRecipeParamsValues[299]);
stActRecipe.stUCF.iCapSorterRobotPickTimeShow.diValue												:=		                STRING_TO_DINT  (aRecipeParamsValues[300]);
stActRecipe.stUCF.iCapSorterRobotVacuumActivationShow.diValue										:=		                STRING_TO_DINT  (aRecipeParamsValues[301]);
stActRecipe.stUCF.iCapSorterRobotVacuumOffShow.diValue						    					:=                      STRING_TO_DINT  (aRecipeParamsValues[302]);
stActRecipe.stUCF.iCapSorterRobotPlaceTimeShow.diValue												:=		                STRING_TO_DINT  (aRecipeParamsValues[303]);
stActRecipe.stUCF.iCapSorterRobotTCP_PlaceOffsetShow.diValue			    						:=				        STRING_TO_DINT  (aRecipeParamsValues[304]);
stActRecipe.stUCF.iCapSorterRobotAccelerationDecelerationShow.diValue	 							:=				        STRING_TO_DINT  (aRecipeParamsValues[305]);
stActRecipe.stUCF.iCapSorterRobotGripperWatchdogShow.diValue			    						:=				        STRING_TO_DINT  (aRecipeParamsValues[306]);
stActRecipe.stUCF.iCapSorterRobotParalaxCorrectionShow.diValue		    							:=			            STRING_TO_DINT  (aRecipeParamsValues[307]);
stActRecipe.stUCF.iCapSorterRobotNumberToolShow.diValue		 										:=				        STRING_TO_DINT  (aRecipeParamsValues[308]);
stActRecipe.stUCF.iCapSorterRobotPickPositionZShow.diValue 											:=			            STRING_TO_DINT  (aRecipeParamsValues[309]);
stActRecipe.stUCF.iCapSorterRobotTCP_Lenght.diValue		 											:=			            STRING_TO_DINT  (aRecipeParamsValues[310]);
stActRecipe.stUCF.iCapSorterRobotProductDiametr.diValue	 											:=			            STRING_TO_DINT  (aRecipeParamsValues[311]);
stActRecipe.stUCF.bCapSorterIntermediateTransporterEnableShow.bValue								:=		                STRING_TO_BOOL  (aRecipeParamsValues[312]);
stActRecipe.stUCF.iCapSorterIntermediateTransporterAutoSpeedShow.diValue							:=		                STRING_TO_DINT  (aRecipeParamsValues[313]);
stActRecipe.stUCF.iCapSorterIntermediateTransporterManualSpeedShow.diValue							:=	                    STRING_TO_DINT  (aRecipeParamsValues[314]);
stActRecipe.stUCF.iCapSorterIntermediateTransporterEmptyingSpeedShow.diValue						:=		                STRING_TO_DINT  (aRecipeParamsValues[315]);
stActRecipe.stUCF.iCapSorterIntermediateTransporterDelayCountTimeShow.diValue						:=	                    STRING_TO_DINT  (aRecipeParamsValues[316]);
stActRecipe.stUCF.iCapSorterIntermediateTransporterReverseTimeShow.diValue							:=	                    STRING_TO_DINT  (aRecipeParamsValues[317]);
stActRecipe.stUCF.udiCapSorterIntermediateTransporterTimeProductOnSensorShow.udiValue 				:=	            		STRING_TO_UDINT (aRecipeParamsValues[318]);
stActRecipe.stUCF.lrCapSorterIntermediateTransporterWheelAngleShow.lrValue							:=    	        		STRING_TO_LREAL (aRecipeParamsValues[319]);
stActRecipe.stUCF.bCapSorterIntermediateBrushEnableShow.bValue			 	    					:=                      STRING_TO_BOOL  (aRecipeParamsValues[320]);
stActRecipe.stUCF.iCapSorterIntermediateBrushAutoSpeedShow.diValue		 	    					:=                      STRING_TO_DINT  (aRecipeParamsValues[321]);
stActRecipe.stUCF.iCapSorterIntermediateBrushManualSpeedShow.diValue		  						:=                      STRING_TO_DINT  (aRecipeParamsValues[322]);
stActRecipe.stUCF.iCapSorterIntermediateBrushEmptyingSpeedShow.diValue	 	    					:=                      STRING_TO_DINT  (aRecipeParamsValues[323]);
stActRecipe.stUCF.lrCapSorterIntermediateBrushPositionHeightSVShow.lrValue 							:=						STRING_TO_LREAL (aRecipeParamsValues[324]);
stActRecipe.stUCF.bCapSorterBrush1OnWheelEnableShow.bValue			  								:=			            STRING_TO_BOOL  (aRecipeParamsValues[325]);
stActRecipe.stUCF.iCapSorterBrush1OnWheelAutoSpeedShow.diValue		  								:=			            STRING_TO_DINT  (aRecipeParamsValues[326]);
stActRecipe.stUCF.iCapSorterBrush1OnWheelManualSpeedShow.diValue		     						:=					    STRING_TO_DINT  (aRecipeParamsValues[327]);
stActRecipe.stUCF.iCapSorterBrush1OnWheelEmptyingSpeedShow.diValue	  								:=			            STRING_TO_DINT  (aRecipeParamsValues[328]);
stActRecipe.stUCF.lrCapSorterBrush1OnWheelPositionHeightSVShow.lrValue   							:=				        STRING_TO_LREAL (aRecipeParamsValues[329]);
stActRecipe.stUCF.bCapSorterBrush2OnWheelEnableShow.bValue			 								:=			            STRING_TO_BOOL  (aRecipeParamsValues[330]);
stActRecipe.stUCF.iCapSorterBrush2OnWheelAutoSpeedShow.diValue		 								:=			            STRING_TO_DINT  (aRecipeParamsValues[331]);
stActRecipe.stUCF.iCapSorterBrush2OnWheelManualSpeedShow.diValue	      							:=				        STRING_TO_DINT  (aRecipeParamsValues[332]);
stActRecipe.stUCF.iCapSorterBrush2OnWheelEmptyingSpeedShow.diValue	   								:=			            STRING_TO_DINT  (aRecipeParamsValues[333]);
stActRecipe.stUCF.lrCapSorterBrush2OnWheelPositionHeightSVShow.lrValue   							:=				        STRING_TO_LREAL (aRecipeParamsValues[334]);
stActRecipe.stUCF.bCapSorterFeederEnableShow.bValue													:=	                    STRING_TO_BOOL  (aRecipeParamsValues[335]);
stActRecipe.stUCF.bCapSorterFeederEnableTubeError.bValue											:=				        STRING_TO_BOOL  (aRecipeParamsValues[336]);
stActRecipe.stUCF.lrCapSorterFeederMover1InputPositionShow.lrValue									:=			            STRING_TO_LREAL (aRecipeParamsValues[337]);
stActRecipe.stUCF.lrCapSorterFeederMover2InputPositionShow.lrValue									:=			            STRING_TO_LREAL (aRecipeParamsValues[338]);
stActRecipe.stUCF.lrCapSorterFeederMover1OutputPositionShow.lrValue									:=			            STRING_TO_LREAL (aRecipeParamsValues[339]);
stActRecipe.stUCF.lrCapSorterFeederMover2OutputPositionShow.lrValue									:=			            STRING_TO_LREAL (aRecipeParamsValues[340]);
stActRecipe.stUCF.lrCapSorterFeederSlotDistanceShow.lrValue											:=			            STRING_TO_LREAL (aRecipeParamsValues[341]);
stActRecipe.stUCF.lrCapSorterFeederMoverSpeedShow.lrValue											:=		                STRING_TO_LREAL (aRecipeParamsValues[342]);
stActRecipe.stUCF.lrCapSorterFeederMoverAccelerationShow.lrValue    								:=			            STRING_TO_LREAL (aRecipeParamsValues[343]);
stActRecipe.stUCF.lrCapSorterFeederMoveJerkShow.lrValue												:=		                STRING_TO_LREAL (aRecipeParamsValues[344]);
stActRecipe.stUCF.bCapSorterPreScrewerEnableShow.bValue												:=		                STRING_TO_BOOL  (aRecipeParamsValues[345]);
stActRecipe.stUCF.bCapSorterPreScrewerPicker1EnableShow.bValue           							:=				        STRING_TO_BOOL  (aRecipeParamsValues[346]);
stActRecipe.stUCF.bCapSorterPreScrewerPicker2EnableShow.bValue           							:=				        STRING_TO_BOOL  (aRecipeParamsValues[347]);
stActRecipe.stUCF.bCapSorterPreScrewerPicker3EnableShow.bValue          							:=				        STRING_TO_BOOL  (aRecipeParamsValues[348]);
stActRecipe.stUCF.bCapSorterPreScrewerPicker4EnableShow.bValue          							:=	                    STRING_TO_BOOL  (aRecipeParamsValues[349]);
stActRecipe.stUCF.lrCapSorterPreScrewerPickZPositionShow.lrValue									:=      		        STRING_TO_LREAL (aRecipeParamsValues[350]);
stActRecipe.stUCF.lrCapSorterPreScrewerCatcherReleseShow.lrValue									:=      		        STRING_TO_LREAL (aRecipeParamsValues[351]);
stActRecipe.stUCF.lrCapSorterPreScrewerCapCatcherZPositionShow.lrValue								:=  		            STRING_TO_LREAL (aRecipeParamsValues[352]);
stActRecipe.stUCF.lrCapSorterPreScrewerTopZPositionShow.lrValue										:=  		            STRING_TO_LREAL (aRecipeParamsValues[353]);
stActRecipe.stUCF.lrCapSorterPreScrewerCartesianCatchZPositionShow.lrValue							:=  		            STRING_TO_LREAL (aRecipeParamsValues[354]);
stActRecipe.stUCF.lrCapSorterPreScrewerStrawCatcherZPositionShow.lrValue							:=	     		        STRING_TO_LREAL (aRecipeParamsValues[355]);
stActRecipe.stUCF.LrCapSorterPreScrewerCheckStrawCatcherActuatorZPosition.lrValue 					:=	 		        	STRING_TO_LREAL (aRecipeParamsValues[356]);
stActRecipe.stUCF.lrCapSorterPreScrewerScrewerStartZPositionShow.lrValue							:=	     		        STRING_TO_LREAL (aRecipeParamsValues[357]);
stActRecipe.stUCF.lrCapSorterPreScrewerGripperOpenPositionShow.lrValue								:=	                    STRING_TO_LREAL (aRecipeParamsValues[358]);
stActRecipe.stUCF.lrCapSorterPreScrewerPlaceZPositionShow.lrValue									:=	                    STRING_TO_LREAL (aRecipeParamsValues[359]);
stActRecipe.stUCF.lrCapSorterPreScrewerBendingDistanceShow.lrValue              					:=                      STRING_TO_LREAL (aRecipeParamsValues[360]);
stActRecipe.stUCF.lrCapSorterPreScrewerStrawInsertDistance.lrValue              					:=                      STRING_TO_LREAL (aRecipeParamsValues[361]);
stActRecipe.stUCF.lrCapSorterPreScrewerPickXMover1PositionShow.lrValue          					:=                      STRING_TO_LREAL (aRecipeParamsValues[362]);
stActRecipe.stUCF.lrCapSorterPreScrewerPickXMover2PositionShow.lrValue          					:=                      STRING_TO_LREAL (aRecipeParamsValues[363]);
stActRecipe.stUCF.lrCapSorterPreScrewerPlaceXPositionShow.lrValue		        					:=                      STRING_TO_LREAL (aRecipeParamsValues[364]);
stActRecipe.stUCF.lrCapSorterPreScrewerScrewFindingShow.lrValue	                					:=              		STRING_TO_LREAL (aRecipeParamsValues[365]);
stActRecipe.stUCF.lrCapSorterPreScrewerScrewDistanceShow.lrValue                					:=               		STRING_TO_LREAL (aRecipeParamsValues[366]);
stActRecipe.stUCF.lrCapSorterPreScrewerPickerSpeedShow.lrValue		            					:=                    	STRING_TO_LREAL (aRecipeParamsValues[367]);
stActRecipe.stUCF.lrCapSorterPreScrewerPickerAccelerationShow.lrValue	        					:=                      STRING_TO_LREAL (aRecipeParamsValues[368]);
stActRecipe.stUCF.lrCapSorterPreScrewerPickerJerkShow.lrValue			        					:=                      STRING_TO_LREAL (aRecipeParamsValues[369]);
stActRecipe.stUCF.lrCapSorterPreScrewerCatcherSpeedShow.lrValue		            					:=                   	STRING_TO_LREAL (aRecipeParamsValues[370]);
stActRecipe.stUCF.lrCapSorterPreScrewerCatcherAccelerationShow.lrValue          					:=                      STRING_TO_LREAL (aRecipeParamsValues[371]);
stActRecipe.stUCF.lrCapSorterPreScrewerCatcherJerkShow.lrValue		            					:=                     	STRING_TO_LREAL (aRecipeParamsValues[372]);
stActRecipe.stUCF.lrCapSorterPreScrewerScrewSpeedShow.lrValue			        					:=                      STRING_TO_LREAL (aRecipeParamsValues[373]);
stActRecipe.stUCF.lrCapSorterPreScrewerScrewAccelerationShow.lrValue	        					:=                      STRING_TO_LREAL (aRecipeParamsValues[374]);
stActRecipe.stUCF.lrCapSorterPreScrewerScrewJerkShow.lrValue			        					:=                      STRING_TO_LREAL (aRecipeParamsValues[375]);
stActRecipe.stUCF.lrCapSorterPreScrewerCatcherCatchingPositionShow.lrValue      					:=                      STRING_TO_LREAL (aRecipeParamsValues[376]);
stActRecipe.stUCF.lrCapSorterPreScrewerCatcherPlacePositionShow.lrValue	        					:=                      STRING_TO_LREAL (aRecipeParamsValues[377]);
stActRecipe.stUCF.lrCapSorterPreScrewerCatcherHightSVShow.lrValue			    					:=                      STRING_TO_LREAL (aRecipeParamsValues[378]);
stActRecipe.stUCF.bCapSorterPreScrewerBottleCatcherEnableShow.bValue		    					:=                      STRING_TO_BOOL  (aRecipeParamsValues[379]);
stActRecipe.stUCF.lrCapSorterPreScrewerBottleCatch1OpenValueShow.lrValue	    					:=                      STRING_TO_LREAL (aRecipeParamsValues[380]);
stActRecipe.stUCF.lrCapSorterPreScrewerBottleCatch1CloseValueShow.lrValue	    					:=                      STRING_TO_LREAL (aRecipeParamsValues[381]);
stActRecipe.stUCF.lrCapSorterPreScrewerBottleCatch2OpenValueShow.lrValue	    					:=                      STRING_TO_LREAL (aRecipeParamsValues[382]);
stActRecipe.stUCF.lrCapSorterPreScrewerBottleCatch2CloseValueShow.lrValue	    					:=                      STRING_TO_LREAL (aRecipeParamsValues[383]);
stActRecipe.stUCF.lrCapSorterPreScrewerBottleCatch3OpenValueShow.lrValue	    					:=                      STRING_TO_LREAL (aRecipeParamsValues[384]);
stActRecipe.stUCF.lrCapSorterPreScrewerBottleCatch3CloseValueShow.lrValue	    					:=                      STRING_TO_LREAL (aRecipeParamsValues[385]);
stActRecipe.stUCF.lrCapSorterPreScrewerBottleCatch4OpenValueShow.lrValue	                      	:=						STRING_TO_LREAL (aRecipeParamsValues[386]);
stActRecipe.stUCF.lrCapSorterPreScrewerBottleCatch4CloseValueShow.lrValue	                      	:= 						STRING_TO_LREAL (aRecipeParamsValues[387]);
stActRecipe.stUCF.lrCapSorterPreScrewerBottleCatchToleranceValueShow.lrValue                      	:= 						STRING_TO_LREAL (aRecipeParamsValues[388]);
stActRecipe.stUCF.lrCapSorterPreScrewerCatchAngleOpenSV.lrValue                       				:= 						STRING_TO_LREAL (aRecipeParamsValues[389]);
stActRecipe.stUCF.lrCapSorterPreScrewerWaitInPlaceTimeShow.lrValue                                	:= 						STRING_TO_LREAL (aRecipeParamsValues[390]);
stActRecipe.stUCF.bCapSorterPreScrewerCatchAngleOpenEnaShow.bValue                                	:= 						STRING_TO_BOOL  (aRecipeParamsValues[391]);
stActRecipe.stUCF.bCapSorterPreScrewerPoundedInCap.bValue                       					:= 						STRING_TO_BOOL  (aRecipeParamsValues[392]);
stActRecipe.stUCF.lrCapSorterBottleHightShow.lrValue		                                      	:= 						STRING_TO_LREAL (aRecipeParamsValues[393]);
stActRecipe.stUCF.lrCapSorterBottleNeckHightShow.lrValue	                                      	:= 						STRING_TO_LREAL (aRecipeParamsValues[394]);
stActRecipe.stUCF.lrCapSorterCapHightShow.lrValue			                                      	:= 						STRING_TO_LREAL (aRecipeParamsValues[395]);
stActRecipe.stUCF.lrCapSorterCapNeckHightShow.lrValue		                                      	:= 						STRING_TO_LREAL (aRecipeParamsValues[396]);
stActRecipe.stUCF.lrCapSorterSpare1.lrValue                											:= 						STRING_TO_LREAL (aRecipeParamsValues[397]);
stActRecipe.stUCF.lrCapSorterSpare2.lrValue                											:= 						STRING_TO_LREAL (aRecipeParamsValues[398]);
stActRecipe.stUCF.lrCapSorterSpare3.lrValue                											:= 						STRING_TO_LREAL (aRecipeParamsValues[399]);
stActRecipe.stUCF.lrCapSorterSpare4.lrValue                											:= 						STRING_TO_LREAL (aRecipeParamsValues[400]);
stActRecipe.stUCF.lrCapSorterSpare5.lrValue                											:= 						STRING_TO_LREAL (aRecipeParamsValues[401]);
stActRecipe.stUCF.lrCapSorterSpare6.lrValue                											:= 						STRING_TO_LREAL (aRecipeParamsValues[402]);
stActRecipe.stUCF.lrCapSorterSpare7.lrValue                											:= 						STRING_TO_LREAL (aRecipeParamsValues[403]);
stActRecipe.stUBF.iBottleSorterProductTypeShow.diValue                                            	:= 						STRING_TO_DINT  (aRecipeParamsValues[404]);
stActRecipe.stUBF.uiBottleSorterIndexShow.diValue		                               				:= 						STRING_TO_DINT  (aRecipeParamsValues[405]);
stActRecipe.stUBF.bBottleSorterHopperTransporterEnableShow.bValue								  	:= 						STRING_TO_BOOL  (aRecipeParamsValues[406]);
stActRecipe.stUBF.iBottleSorterHopperConveyorRunningSpeedSVShow.diValue							  	:= 						STRING_TO_DINT  (aRecipeParamsValues[407]);
stActRecipe.stUBF.iBottleSorterHopperConveyorEmptyingSpeedSVShow.diValue							:= 						STRING_TO_DINT  (aRecipeParamsValues[408]);
stActRecipe.stUBF.iBottleSorterDistanceToFindElementOnTransferConveyorLimitRunningSVShow.diValue	:= 						STRING_TO_DINT  (aRecipeParamsValues[409]);
stActRecipe.stUBF.iBottleSorterDistanceToFindElementOnTransferConveyorLimitEmptyingSVShow.diValue 	:= 						STRING_TO_DINT  (aRecipeParamsValues[410]);
stActRecipe.stUBF.bBottleSorterTransferTransporterEnableShow.bValue								  	:= 						STRING_TO_BOOL  (aRecipeParamsValues[411]);
stActRecipe.stUBF.iBottleSorterTransferConveyorRunningSpeedSVShow.diValue						  	:= 						STRING_TO_DINT  (aRecipeParamsValues[412]);
stActRecipe.stUBF.iBottleSorterTransferConveyorEmptyingSpeedSVShow.diValue						  	:=						STRING_TO_DINT  (aRecipeParamsValues[413]);
stActRecipe.stUBF.iBottleSorterDistanceToFindElementOnSupplyConveyorDownstairsLimitSVShow.diValue 	:= 						STRING_TO_DINT  (aRecipeParamsValues[414]);
stActRecipe.stUBF.bBottleSorterSupplyTransporterEnableShow.bValue			                      	:= 						STRING_TO_BOOL  (aRecipeParamsValues[415]);
stActRecipe.stUBF.uiBottleSorterSupplyTransporterRunningSpeedSVShow.udiValue                      	:= 						STRING_TO_UDINT (aRecipeParamsValues[416]);
stActRecipe.stUBF.uiBottleSorterSupplyTransporterEmptingSpeedSVShow.udiValue                      	:= 						STRING_TO_UDINT (aRecipeParamsValues[417]);
stActRecipe.stUBF.lrBottleSorterModuloMoveOffsetSVShow.lrValue				                      	:= 						STRING_TO_LREAL (aRecipeParamsValues[418]);
stActRecipe.stUBF.iBottleSorterSensorsCountFirstConditionSVShow.diValue	                          	:= 						STRING_TO_DINT  (aRecipeParamsValues[419]);
stActRecipe.stUBF.iBottleSorterSupplyTimeFirstConditionSVShow.diValue		                      	:= 						STRING_TO_DINT  (aRecipeParamsValues[420]);
stActRecipe.stUBF.iBottleSorterSensorsCountSecondConditionMinSVShow.diValue	                      	:= 						STRING_TO_DINT  (aRecipeParamsValues[421]);
stActRecipe.stUBF.iBottleSorterSensorsCountSecondConditionMaxSVShow.diValue	                      	:= 						STRING_TO_DINT  (aRecipeParamsValues[422]);
stActRecipe.stUBF.iBottleSorterSupplyTimeSecondConditionSVShow.diValue		                      	:= 						STRING_TO_DINT  (aRecipeParamsValues[423]);
stActRecipe.stUBF.iBottleSorterSensorsCountThirdConditionSVShow.diValue	                          	:= 						STRING_TO_DINT  (aRecipeParamsValues[424]);
stActRecipe.stUBF.iBottleSorterSupplyTimeThirdConditionSVShow.diValue		                      	:= 						STRING_TO_DINT  (aRecipeParamsValues[425]);
stActRecipe.stUBF.bBottleSorterWeelEnableShow.bValue			                       				:= 						STRING_TO_BOOL  (aRecipeParamsValues[426]);
stActRecipe.stUBF.lrBottleSorterWheelSpeedSVShow.lrValue			                             	:= 						STRING_TO_LREAL (aRecipeParamsValues[427]);
stActRecipe.stUBF.lrBottleSorterWheelEmptyingSpeedSVShow.lrValue	                              	:= 						STRING_TO_LREAL (aRecipeParamsValues[428]);
stActRecipe.stUBF.bBottleSorterBrushEnableShow.bValue			   									:= 						STRING_TO_BOOL  (aRecipeParamsValues[429]);
stActRecipe.stUBF.lrBottleSorterBrushHeightPositionSVShow.lrValue                                 	:= 						STRING_TO_LREAL (aRecipeParamsValues[430]);
stActRecipe.stUBF.iBottleSorterBrushRunningSpeedSVShow.diValue	                                  	:= 						STRING_TO_DINT  (aRecipeParamsValues[431]);
stActRecipe.stUBF.iBottleSorterBrushEmptyingSpeedSVShow.diValue	                                  	:= 						STRING_TO_DINT  (aRecipeParamsValues[432]);
stActRecipe.stUBF.bBottleSorterRobotEnableShow.bValue	                            				:= 						STRING_TO_BOOL  (aRecipeParamsValues[433]);
stActRecipe.stUBF.nBottleSorterRobotRecipeId.udiValue		                                		:= 						STRING_TO_UDINT (aRecipeParamsValues[434]);
stActRecipe.stUBF.lrBottleSorterRemainingTimeToSuctionShow.lrValue                                	:= 						STRING_TO_LREAL (aRecipeParamsValues[435]);
stActRecipe.stUBF.lrBottleSorterSuckerSuctionTimeShow.lrValue		                              	:= 						STRING_TO_LREAL (aRecipeParamsValues[436]);
stActRecipe.stUBF.lrBottleSorterRemainingTimeToRejectShow.lrValue                                 	:= 						STRING_TO_LREAL (aRecipeParamsValues[437]);
stActRecipe.stUBF.lrBottleSorterEjectorPulseShow.lrValue                                        	:= 						STRING_TO_LREAL (aRecipeParamsValues[438]);
stActRecipe.stUBF.lrBottleSorterZPickAboveTheBottleSVShow.lrValue	                              	:= 						STRING_TO_LREAL (aRecipeParamsValues[439]);
stActRecipe.stUBF.lrBottleSorterZPickMoveSVShow.lrValue			                            		:=						STRING_TO_LREAL (aRecipeParamsValues[440]);
stActRecipe.stUBF.lrBottleSorterSafetyHeightSVShow.lrValue		                              		:= 						STRING_TO_LREAL (aRecipeParamsValues[441]);
stActRecipe.stUBF.bBottleSorterRecieverEnableShow.bValue			                              	:= 						STRING_TO_BOOL  (aRecipeParamsValues[442]);
stActRecipe.stUBF.bBottleSorterRecieverSlot1EnableShow.bValue		                              	:= 						STRING_TO_BOOL  (aRecipeParamsValues[443]);
stActRecipe.stUBF.bBottleSorterRecieverSlot2EnableShow.bValue		                              	:= 						STRING_TO_BOOL  (aRecipeParamsValues[444]);
stActRecipe.stUBF.bBottleSorterRecieverSlot3EnableShow.bValue		                				:= 						STRING_TO_BOOL  (aRecipeParamsValues[443]);
stActRecipe.stUBF.lrBottleSorterRecieverHeightPositionSVShow.lrValue                              	:= 						STRING_TO_LREAL (aRecipeParamsValues[444]);
stActRecipe.stUCF.lrCapSorterPreScrewerPickerSpeedWhenScrewerShow.lrValue							:=						STRING_TO_LREAL (aRecipeParamsValues[445]);
stActRecipe.stUBL.bROPPCappingEnableShow.bValue														:=						STRING_TO_BOOL  (aRecipeParamsValues[446]);
stActRecipe.stUBL.bROPPDragEnableShow.bValue	 					                                :=                      STRING_TO_BOOL  (aRecipeParamsValues[447]);
stActRecipe.stUBL.bROPPFeederEnableShow.bValue						                                :=                      STRING_TO_BOOL  (aRecipeParamsValues[448]);
stActRecipe.stUBL.bROPPSlowerEnableShow.bValue	 					                                :=                      STRING_TO_BOOL  (aRecipeParamsValues[449]);
stActRecipe.stUBL.iROPPCapping1ToolShow.diValue 					                                :=      				STRING_TO_DINT 	(aRecipeParamsValues[450]);
stActRecipe.stUBL.iROPPCappingTime2Show.diValue  					                                :=      				STRING_TO_DINT 	(aRecipeParamsValues[451]);
stActRecipe.stUBL.iROPPCappingTimeShow.diValue  					                                :=      				STRING_TO_DINT 	(aRecipeParamsValues[452]);	
stActRecipe.stUBL.iROPPFeederTimeDelayOffShow.diValue 				                                :=      				STRING_TO_DINT 	(aRecipeParamsValues[453]);	
stActRecipe.stUBL.iROPPFeederTimeDelayOnShow.diValue  				                                :=      				STRING_TO_DINT 	(aRecipeParamsValues[454]);
stActRecipe.stUBL.iROPPFeederTimeToEmptySleeveErrorShow.diValue	                                    :=    					STRING_TO_DINT 	(aRecipeParamsValues[455]);
stActRecipe.stUBL.lrROPPCappingHeightPosSVShow.lrValue			                                    :=      				STRING_TO_LREAL (aRecipeParamsValues[456]);
stActRecipe.stUBL.lrROPPCappingVelocitySVShow.lrValue	 			                                :=                      STRING_TO_LREAL (aRecipeParamsValues[457]);
stActRecipe.stUBL.lrROPPDragAccelerationShow.lrValue	 				                            :=                      STRING_TO_LREAL (aRecipeParamsValues[458]);
stActRecipe.stUBL.lrROPPDragDecelerationShow.lrValue	 				                            :=                      STRING_TO_LREAL (aRecipeParamsValues[459]);
stActRecipe.stUBL.lrROPPDragVelocityShow.lrValue	 					                            :=                      STRING_TO_LREAL (aRecipeParamsValues[460]);
stActRecipe.stUBL.lrROPPFeederHeightPosSVShow.lrValue	 			                                :=                      STRING_TO_LREAL (aRecipeParamsValues[461]);
stActRecipe.stUBL.nROPPSlowerVelocitySVShow.udiValue												:=                      STRING_TO_UDINT (aRecipeParamsValues[462]);
END_METHOD

METHOD METH_FindRecipeArrayIndex : DINT
VAR_INPUT
	iSelectedArrayIndex							: INT;
END_VAR
FOR i:=0 TO udiMaxRecipeCount DO
	IF	aRecipeList[i].bUsed AND aRecipeList[i].udiIndex = aRecipeList[iSelectedArrayIndex].udiIndex THEN
		METH_FindRecipeArrayIndex				:= UDINT_TO_DINT(i);
		EXIT;
	END_IF
END_FOR
END_METHOD

METHOD METH_ParseRecipesListStringArray : BOOL
VAR

END_VAR
FOR i := 0 TO udiMaxRecipeCount DO
	aSplit[0] := aRecipeListString[i];
	FOR j:=0 TO 4 DO
		bResultSplit := FindAndSplitChar( sSeparatorChar := '|',  pSrcString := ADR(aSplit[j]), 
	                                      pLeftString    := ADR(aSplit[j]),   nLeftSize  := SIZEOF(aSplit[j]), 
	                                      pRightString   := ADR(aSplit[j+1]), nRightSize := SIZEOF(aSplit[j+1]),
	                                      bSearchFromRight := FALSE );
	    IF NOT bResultSplit THEN
	        EXIT;
	    END_IF
	END_FOR
	aRecipeList[i].bUsed :=STRING_TO_BOOL(aSplit[0]);
	aRecipeList[i].udiIndex :=STRING_TO_UDINT(aSplit[1]);
	aRecipeList[i].wsRecipeCaption :=STRING_TO_WSTRING(aSplit[2]);
	aRecipeList[i].wsRecipeDescription :=STRING_TO_WSTRING(aSplit[3]);
	aRecipeList[i].wsCreateDate :=STRING_TO_WSTRING(aSplit[4]);
END_FOR
END_METHOD

